(* CODESYS project OSCAT NETWORK.library
   Title: OSCAT NETWORK
   Author: Joel Zupancic
   Version: 1.30
   Description: see www.oscat.de for here home
      
      Made changes to use newer version 3 library SysSocket and SysFile.  All code was tested on CoDesys SoftPLC and Schneider Electric PLC with ehternet and file systems and using SoMachine software.
      
      
      IP_CONTROL
      1. Had to Set option for local address reuse in all network cases
        SysSockSetOption(socket, SOCKET_SOL, SOCKET_SO_REUSEADDR, ADR(dint_true), SIZEOF(dint_true));
      2. Had to change NETWORK_BUFFER_LONG_SIZE : UINT := 1999; //Changed from 3999 else socket would not work when reading 
      3. If PORT is zero use port specified by IP_C.C_PORT.
      4. CoDeSys has a bug that does not release the ports on a warm or cold reset.  What this means if you do a reset any function blocks that require binding to the socket to stay open will no longer work.  As of now the only way to clear the port is to recycle the power on the PLC.  
      
      
      TN_FRAMEWORK
      1.  Always Used Port 23. Changed to only use 23 if no port passed via IP_C.PORT
      
      STRING_TO_URL
      1.  Moved VAR_TEMP varible to VAR
      
      WORLD_WEATHER_ICON_OSCAT
      1.  Put [] around dat intial values
      
      YAHOO_WEATHER_ICON_OSCAT
      1.  Put [] around dat intial values
      
      MB_SERVER
      Need to reset the socket after the receive data timed out.  Since there is no code to detect that the Socket is still open you must force the socket closed and wait for the next connection.
      
      Case 10:
      IP_C.R_OBSERVE := TRUE; ( * keine Empfangsueberwachung * )
      
      and 
      
      IF ENABLE = FALSE OR t.Q THEN
          ip_state := BYTE#4; ( * Abmelden * )
         state := 00;
         IP_C.C_ENABLE := FALSE; 
      END_IF;
      
      
      /////////NEED TO FIX//////////////////
      FTP_CLIENT
      1.  Always Used Port 21. Changed to only use 21 if no port as specified in passed URL
   Company: OSCAT

Project tree, tasks and I/O mapping:
  libraries: SysTypes Interfaces, * (System); BASIC, 3.3.3.0 (OSCAT); Standard, * (System); SysSocket23, 3.5.8.0 (System); SysFile23, 3.5.8.0 (System)
  Data types/
    DATA_LOG/
      data type DLOG_CRON_DATA
      data type DLOG_CRON_ELEMENT
      data type DLOG_DATA
      data type DLOG_RETAIN
      data type LOG_CONTROL
      data type PRINTF_DATA
      data type UNI_CIRCULAR_BUFFER_DATA
      data type us_LOG_VIEWPORT
    DATABASE/
      data type MYSQL_COM
      data type MYSQL_INFO
    FILE_SERVER/
      data type FILE_PATH_DATA
      data type FILE_SERVER_DATA
    NET_VAR/
      data type NET_VAR_DATA
    NETWORK/
      data type IP2GEO_DATA
      data type IP_C
      data type IP_FIFO_DATA
      data type NETWORK_BUFFER
      data type NETWORK_BUFFER_SHORT
      data type NW_BUF_LONG
      data type NW_BUF_SHORT
      data type URL
      data type VMAP_DATA
      data type XML_CONTROL
    TELNET_VISION/
      data type us_TN_INPUT_CONTROL
      data type us_TN_INPUT_CONTROL_DATA
      data type us_TN_MENU
      data type us_TN_MENU_POPUP
      data type us_TN_SCREEN
    WEATHER/
      data type WORLD_WEATHER_CUR
      data type WORLD_WEATHER_DATA
      data type WORLD_WEATHER_DAY
      data type YAHOO_WEATHER_DATA
  Global Variables/
    global variables Constants
    global variables Globale_Variablen
  POUs/
    _HARDWARE/
      function block IP_CONTROL [ST]
      function block FILE_SERVER_OLD [ST]
      function block FILE_SERVER [ST]
      function block IP_CONTROL2 [ST]
    CONVERT/
      function block BASE64_DECODE_STR [ST]
      function block BASE64_DECODE_STREAM [ST]
      function block BASE64_ENCODE_STR [ST]
      function block BASE64_ENCODE_STREAM [ST]
      function HTML_DECODE [ST]
      function HTML_ENCODE [ST]
      function IP4_CHECK [ST]
      function IP4_DECODE [ST]
      function IP4_TO_STRING [ST]
      function IS_IP4 [ST]
      function IS_URLCHR [ST]
      function MD5_AUX [ST]
      function block MD5_CRAM_AUTH [ST]
      function block MD5_STR [ST]
      function block MD5_STREAM [ST]
      function MD5_TO_STRH [ST]
      function block RC4_CRYPT_STREAM [ST]
      function block SHA1_STR [ST]
      function block SHA1_STREAM [ST]
      function SHA1_TO_STRH [ST]
      function STRING_TO_URL [ST]
      function URL_DECODE [ST]
      function URL_ENCODE [ST]
      function URL_TO_STRING [ST]
    DATA_LOG/
      function block DLOG_BOOL [ST]
      function block DLOG_CRON_TAB [ST]
      function block DLOG_DINT [ST]
      function block DLOG_DT [ST]
      function block DLOG_FILE_TO_FTP [ST]
      function block DLOG_FILE_TO_SMTP [ST]
      function block DLOG_REAL [ST]
      function block DLOG_STORE_FILE_CSV [ST]
      function block DLOG_STORE_FILE_HTML [ST]
      function block DLOG_STORE_FILE_XML [ST]
      function block DLOG_STORE_MYSQL [ST]
      function block DLOG_STORE_RRD [ST]
      function block DLOG_STRING [ST]
      function block UNI_CIRCULAR_BUFFER [ST]
    DATABASE/
      function block MYSQL_AUTH [ST]
      function block MYSQL_CONTROL [ST]
    DRIVER/
      function block IRTRANS_DECODE [ST]
      function block IRTRANS_RCV_1 [ST]
      function block IRTRANS_RCV_4 [ST]
      function block IRTRANS_RCV_8 [ST]
      function block IRTRANS_SERVER [ST]
      function block IRTRANS_SND_1 [ST]
      function block IRTRANS_SND_4 [ST]
      function block IRTRANS_SND_8 [ST]
    FILE/
      function block CSV_PARSER_BUF [ST]
      function block CSV_PARSER_FILE [ST]
      function block FILE_BLOCK [ST]
      function FILE_PATH_SPLIT [ST]
      function block INI_PARSER_BUF [ST]
      function block INI_PARSER_FILE [ST]
    HARDWARE/
      function block FILE_SERVER_V2 [ST]
      function block IP_CONTROL_V2 [ST]
      function block IP_CONTROL2_V2 [ST]
    NET_VAR/
      function block NET_VAR_BOOL8 [ST]
      function block NET_VAR_BUFFER [ST]
      function block NET_VAR_CONTROL [ST]
      function block NET_VAR_DWORD8 [ST]
      function block NET_VAR_REAL8 [ST]
      function block NET_VAR_STRING [ST]
      function block NET_VAR_X8 [ST]
    NETWORK/
      function block DNS_CLIENT [ST]
      function block DNS_DYN [ST]
      function block DNS_REV_CLIENT [ST]
      function block FTP_CLIENT [ST]
      function block GET_WAN_IP [ST]
      function block HTTP_GET [ST]
      function block IP2GEO [ST]
      function block IP_FIFO [ST]
      function block LOG_MSG [ST]
      function block LOG_VIEWPORT [ST]
      function block MB_CLIENT [ST]
      function block MB_SERVER [ST]
      function block MB_SERVER_1 [ST]
      function block MB_VMAP [ST]
      function block PRINT_SF [ST]
      function block READ_HTTP [ST]
      function block SMTP_CLIENT [ST]
      function block SNTP_CLIENT [ST]
      function block SNTP_SERVER [ST]
      function block SPIDER_ACCESS [ST]
      function block SYS_LOG [ST]
      function block TELNET_LOG [ST]
      function block TELNET_PRINT [ST]
      function block XML_READER [ST]
    OTHER/
      function ELEMENT_COUNT [ST]
      function ELEMENT_GET [ST]
      function NETWORK_VERSION [ST]
    TELNET_VISION/
      function block TN_FRAMEWORK [ST]
      function block TN_INPUT_CONTROL [ST]
      function block TN_INPUT_EDIT_LINE [ST]
      function block TN_INPUT_MENU_BAR [ST]
      function block TN_INPUT_MENU_POPUP [ST]
      function block TN_INPUT_SELECT_POPUP [ST]
      function block TN_INPUT_SELECT_TEXT [ST]
      function block TN_RECEIVE [ST]
      function block TN_SC_ADD_SHADOW [ST]
      function block TN_SC_AREA_RESTORE [ST]
      function block TN_SC_AREA_SAVE [ST]
      function block TN_SC_BOX [ST]
      function block TN_SC_FILL [ST]
      function block TN_SC_LINE [ST]
      function block TN_SC_READ_ATTR [ST]
      function block TN_SC_READ_CHAR [ST]
      function TN_SC_SHADOW_ATTR [ST]
      function block TN_SC_VIEWPORT [ST]
      function block TN_SC_WRITE [ST]
      function block TN_SC_WRITE_ATTR [ST]
      function block TN_SC_WRITE_C [ST]
      function block TN_SC_WRITE_CHAR [ST]
      function block TN_SC_WRITE_EOS [ST]
      function TN_SC_XY2_ERROR [ST]
      function TN_SC_XY_ERROR [ST]
      function block TN_SEND_ROWS [ST]
    WEATHER/
      function block MOON_PHASE [ST]
      function block WORLD_WEATHER [ST]
      function block WORLD_WEATHER_DESC_GE [ST]
      function block WORLD_WEATHER_ICON_OSCAT [ST]
      function block YAHOO_WEATHER [ST]
      function block YAHOO_WEATHER_DESC_GE [ST]
      function block YAHOO_WEATHER_ICON_OSCAT [ST]
    DEMO/
      OLD/
        program INI_PARSER_FILE_DEMO_OLD [ST]
        program INI_PARSER_BUF_DEMO_OLD [ST]
      global variables GVL_DEMO
      Need Fixing/
        program IRTRANS_DEMO [CFC]
      WORKING/
        program INI_PARSER_BUF_DEMO [ST]
        program INI_PARSER_FILE_DEMO [ST]
        program _ECHO_TEST_DEMO [CFC]
        program CSV_PARSER_FILE_DEMO [ST]
        program TN_VISION_DEMO_1 [ST]
        program RC4_CRYPT_DEMO [CFC]
        program FILE_BLOCK_DEMO [CFC]
        program GET_WAN_IP_DEMO [CFC]
        program BASE64_DEMO [CFC]
        program DNS_SNTP_SYSLOG_DEMO [CFC]
        program DLOG_RRD_DEMO [CFC]
        program CSV_PARSER_BUF_DEMO [ST]
        program DNS_DYN_DEMO [CFC]
        program TN_VISION_DEMO_2 [ST]
        program YAHOO_WEATHER_DEMO [CFC]
        program MB_CLIENT_DEMO [CFC]
        program TELNET_LOG_DEMO [CFC]
        program SHA1_MD5_DEMO [CFC]
        program IP2GEO_DEMO [CFC]
        program FTP_CLIENT_DEMO [CFC]
        program MD5_CRAM_AUTH_DEMO [CFC]
        program DNS_CLEINT_DEMO [CFC]
        program TELNET_PRINT_DEMO [CFC]
        program HTTP_DEMO [CFC]
        program WORLD_WEATHER_DEMO [CFC]
        program MB_SERVER_DEMO [CFC]
        program SMTP_CLIENT_DEMO [CFC]
        program DNS_REV_DEMO [CFC]
      Need_Testing/
        program DLOG_FILE_CSV_FTP_DEMO [CFC]
        program DLOG_FILE_CSV_DEMO [CFC]
        program NET_VAR_SLAVE_DEMO [CFC]
        program DLOG_FILE_CSV_SMTP_DEMO [CFC]
        program SPIDER_DEMO [CFC]
        program DLOG_FILE_HTML_DEMO [CFC]
        program NET_VAR_MASTER_DEMO [CFC]
        program DLOG_MYSQL_DEMO [CFC]
        program DLOG_FILE_XML_DEMO [CFC]
  Visualizations/
*)

// Data types/DATA_LOG/DLOG_CRON_DATA
TYPE DLOG_CRON_DATA :
STRUCT
	CE : ARRAY [0..5] OF DLOG_CRON_ELEMENT;
END_STRUCT
END_TYPE

// Data types/DATA_LOG/DLOG_CRON_ELEMENT
TYPE DLOG_CRON_ELEMENT :
STRUCT
	ELEMENTS : ARRAY [0..59] OF BOOL;
	VALUE : INT;
	VALUE_MIN : INT;
	VALUE_MAX : INT;
	ALL_SELECTED : BOOL;
END_STRUCT
END_TYPE

// Data types/DATA_LOG/DLOG_DATA
TYPE DLOG_DATA :
STRUCT
	STORE_TYPE : BYTE;
	ADD_COM : INT;
	ADD_DATA_REQ : BOOL;
	CLOCK_TRIG : BOOL;
	ID_MAX : USINT;
	DTI : DT;
	UCB : UNI_CIRCULAR_BUFFER_DATA;
	LOAD_TIME_MAX : TIME;
	NEW_FILE : STRING;
	NEW_FILE_SIZE : UDINT;
	NEW_FILE_RTRIG : BOOL;
END_STRUCT
END_TYPE

(* revision history
ks	01. oct. 2010	rev 1.0
	original version

ks	13. may. 2011	rev 1.1
	neues Element: ADD_DATA_REQ

ks	26. jul. 2011	rev 1.2
	neues Element: STORE_TYPE

ks	16. apr. 2012	rev 1.3
	neues Elemente: NEW_FILE_SIZE, ADD_COM
*)

// Data types/DATA_LOG/DLOG_RETAIN
TYPE DLOG_RETAIN :
STRUCT
	FN_REM : STRING;
	COLOR : BOOL;
	HEAD: BOOL;
	TRIG_CNT : UDINT;
	TRIG_CNT_TOTAL : UDINT;
END_STRUCT
END_TYPE

(* revision history
ks	27. oct. 2012	rev 1.0
	original version

*)

// Data types/FILE_SERVER/FILE_PATH_DATA
TYPE FILE_PATH_DATA :
STRUCT
	DRIVE : STRING(3);
	DIRECTORY : STRING(OSCAT_BASIC.STRING_LENGTH);
	FILENAME : STRING;
END_STRUCT
END_TYPE

(* revision history
ks	01. oct. 2010	rev 1.0
	original version
*)

// Data types/FILE_SERVER/FILE_SERVER_DATA
TYPE FILE_SERVER_DATA :
STRUCT
	FILE_OPEN : BOOL;
	FILENAME : STRING;
	MODE : BYTE;
	OFFSET : UDINT;
	FILE_SIZE : UDINT;
	ERROR : BYTE;
END_STRUCT
END_TYPE

(* revision history
ks	05. mai. 2012	rev 1.1
	original version
*)

// Data types/NETWORK/IP2GEO_DATA
TYPE IP2GEO_DATA :
STRUCT
	STATE : BOOL;
	IP4 : DWORD;
	COUNTRY_CODE : STRING(2);
	COUNTRY_NAME : STRING(20);
	REGION_CODE : STRING(2);
	REGION_NAME : STRING(20);
	CITY : STRING(20);
	GEO_LATITUDE : REAL;
	GEO_LONGITUDE : REAL;
	TIME_ZONE_NAME : STRING(20);
	GMT_OFFSET : INT;
	IS_DST : BOOL;
END_STRUCT
END_TYPE

(* revision history
ks	14. aug. 2009	rev 1.0
	original version
*)

// Data types/NETWORK/IP_C
TYPE IP_C :
STRUCT
	C_MODE : BYTE;						(*W Mode: TCP/UCP AKTIV/PASSIV                               *)
	C_PORT : WORD;						(*W Portnummer                                               *)
	C_IP : DWORD;						(*W IP-Adresse gepackt wwxxyyzz = www.xxx.yyy.zzz            *)
	C_STATE : BYTE;						(*R Verbindungsstatus ON/OFF + Flanke ON/OFF                 *)
	C_ENABLE : BOOL;					(*W Freigabe für Connect                                     *)
	R_OBSERVE : BOOL;					(*W Empfang ueberwachen                                      *)
	TIME_RESET : BOOL;					(*W Alle Timer ruecksetzen                                   *)
	ERROR : DWORD;					(*R vvwwxxyy (vv = CON_ERROR, ww = SEN_ERROR, xx = REC_ERROR *)
	FIFO : IP_FIFO_DATA;					(*I IP FIFO Struktur                                         *)
	MAILBOX : ARRAY [1..16] OF BYTE;	(*I Mailbox: Datenbereich für Bausteindatenaustausch         *)
END_STRUCT
END_TYPE

(* revision history
ks	18. oct. 2008	rev 1.0
	original version
*)

// Data types/NETWORK/IP_FIFO_DATA
TYPE IP_FIFO_DATA :
STRUCT
	X : ARRAY [1..128] OF BYTE; 	(* IP_ID FIFO Speicher          *)
	Y : ARRAY [1..128] OF BYTE; 	(* IP_ID Zähler                 *)
	ID : BYTE;					(* höchste vergabene id         *)
	MAX_ID : BYTE;				(* maximal Anmeldungen pro ID   *)
	INIT : BOOL;					(* Initialisierung durchgeführt *)
	EMPTY : BOOL;				(* FIFO leer                    *)
	FULL : BOOL;					(* FIFO voll                    *)
	TOP : INT;					(* maximale anzahl in FIFO      *)
	NW : INT;					(* Schreibzeiger                *)
	NR : INT;						(* Lesezeiger                   *)
END_STRUCT
END_TYPE

(* revision history
ks	18. oct. 2008	rev 1.0
	original version
*)

// Data types/DATA_LOG/LOG_CONTROL
TYPE LOG_CONTROL :
STRUCT
	NEW_MSG : STRING(LOG_SIZE); (* neue Nachricht für den Datenbuffer *)
	NEW_MSG_OPTION : DWORD;
	LEVEL : BYTE;
	SIZE : INT := LOG_MAX; (* Anzahl der Strings im LOG_DATA *)
	RESET : BOOL; (* Nachrichtenbuffer löschen *)
	PRINTF : PRINTF_DATA; (* Array PRINTF Parameter *)
	MSG : ARRAY [0..LOG_MAX] OF STRING(LOG_SIZE); (* Array Message *)
	MSG_OPTION : ARRAY [0..LOG_MAX] OF DWORD; (* Array Options *)
	UPDATE_COUNT : UINT; (* Updatezähler *)
	IDX : INT; (* aktueller Nachrichten-Index *)
	RING_MODE : BOOL; (* Bufferüberlauf erkannt *)
END_STRUCT
END_TYPE

(* revision history
ks	18. oct. 2008	rev 1.0
	original version

ks	17..may. 2011	rev 1.1
	ENABLE entfernt

*)

// Data types/DATABASE/MYSQL_COM
TYPE MYSQL_COM :
STRUCT
	S_BUF : NETWORK_BUFFER;
	R_BUF : NETWORK_BUFFER;
	SQL_CON : BOOL;
	SQL_URL : STRING(OSCAT_BASIC.STRING_LENGTH);
	SQL_PACKET_NO : BYTE;
	TIMEOUT : TIME;
	DNS_IP4 : DWORD;
	SQL_RCV_STATE : BYTE;
	ERROR_C : DWORD;
	ERROR_T : BYTE;
END_STRUCT
END_TYPE

(* revision history
ks	27. oct. 2012	rev 1.0
	original version
*)

// Data types/DATABASE/MYSQL_INFO
TYPE MYSQL_INFO :
STRUCT
	SERVER_PROTOCOL_VERSION : BYTE;
	SERVER_CAPABILITIES : WORD;
	SERVER_STATUS : WORD;
	SERVER_LANGUAGE : BYTE;
	SQL_CONNECTED : BOOL;
	SQL_ERROR : STRING(OSCAT_BASIC.STRING_LENGTH);
END_STRUCT
END_TYPE

(* revision history
ks	27. oct. 2012	rev 1.0
	original version
*)

// Data types/NET_VAR/NET_VAR_DATA
TYPE NET_VAR_DATA :
STRUCT
	CYCLE : UDINT;
	STATE : BYTE;
	INDEX : INT;
	ID_MAX : USINT;
	ERROR_ID : BYTE;
	BUF_SIZE : UINT;
	S_BUF : NETWORK_BUFFER;
	R_BUF : NETWORK_BUFFER;
END_STRUCT
END_TYPE

(* revision history
ks	01. feb. 2011	rev 1.0
	original version
*)

// Data types/NETWORK/NETWORK_BUFFER
TYPE NETWORK_BUFFER :
STRUCT
	SIZE : UINT;
	BUFFER : NW_BUF_LONG;
END_STRUCT
END_TYPE

(* revision history
ks	01. 01. 2009	rev 1.0
	original version
*)

// Data types/NETWORK/NETWORK_BUFFER_SHORT
TYPE NETWORK_BUFFER_SHORT :
STRUCT
	SIZE : UINT;
	BUFFER : NW_BUF_SHORT;
END_STRUCT
END_TYPE

(* revision history
ks	01. 01. 2009	rev 1.0
	original version
*)

// Data types/NETWORK/NW_BUF_LONG
TYPE
	NW_BUF_LONG  : ARRAY[0..NETWORK_BUFFER_LONG_SIZE] OF BYTE;
END_TYPE

(* revision history
ks	01. 01. 2009	rev 1.0
	original version
*)

// Data types/NETWORK/NW_BUF_SHORT
TYPE
	NW_BUF_SHORT : ARRAY[0..NETWORK_BUFFER_SHORT_SIZE] OF BYTE;
END_TYPE

(* revision history
ks	01. 01. 2009	rev 1.0
	original version
*)

// Data types/DATA_LOG/PRINTF_DATA
TYPE PRINTF_DATA : ARRAY [1..11]  OF STRING(LOG_SIZE);
END_TYPE

(* revision history
ks	18. oct. 2008
	original version
*)

// Data types/DATA_LOG/UNI_CIRCULAR_BUFFER_DATA
TYPE UNI_CIRCULAR_BUFFER_DATA :
STRUCT
	D_MODE : INT;
	D_HEAD : WORD;
	D_STRING : STRING(OSCAT_BASIC.STRING_LENGTH);
	D_REAL : REAL;
	D_DWORD : DWORD;
	BUF_SIZE : UINT;
	BUF_COUNT : UINT;
	BUF_USED : USINT;
	BUF : NW_BUF_LONG;
	_GetStart : UINT;
	_GetEnd : UINT;
	_Last : UINT;
	_First : UINT;
END_STRUCT
END_TYPE

(* revision history
ks	01. oct. 2010	rev 1.0
	original version
*)

// Data types/NETWORK/URL
TYPE URL :
STRUCT
	PROTOCOL : STRING(10);
	USER : STRING(32);
	PASSWORD : STRING(32);
	DOMAIN : STRING(80);
	PORT : WORD;
	PATH : STRING(80);
	QUERY : STRING(OSCAT_BASIC.STRING_LENGTH);
	ANCHOR : STRING(40);
	HEADER : STRING(160);
END_STRUCT
END_TYPE

(* revision history
hm	18. oct. 2008 v1.0
	original version

ks	01.oct.2010 v1.1
	new header element and string size
*)

// Data types/DATA_LOG/us_LOG_VIEWPORT
TYPE us_LOG_VIEWPORT :
STRUCT
	LINE_ARRAY : ARRAY [1..40] OF INT;
	COUNT : INT; (* Anzahl der sichtbaren Nachtrichten *)
	UPDATE_COUNT : UINT; (* Updatezähler *)
	MOVE_TO_X : INT; (* Steuerung der Nachrichtenanzeige *)
	UPDATE : BOOL; (* Daten wurden geändert -> neuzeichnen *)
END_STRUCT
END_TYPE

(* revision history
ks	18. oct. 2008	rev 1.0
	original version
*)

// Data types/TELNET_VISION/us_TN_INPUT_CONTROL
TYPE us_TN_INPUT_CONTROL :
STRUCT
	bo_Enable: BOOL; (* Bearbeitung freigeben/sperren *)
	bo_Update_all: BOOL; (* All Elemente neu zeichnen *)
	bo_Reset_Fokus: BOOL; (* Fokus auf 1. Element setzen *)
	in_Focus_at: INT; (* Controlelement mit aktivem Fokus *)
	in_Count: INT; (* Anzahl der benutzen Control-Elemente *)
	in_ToolTip_X: INT; (* Tooltip Text X-Offset *)
	in_ToolTip_Y: INT; (* Tooltip Text Y-Offset *)
	by_ToolTip_Attr: BYTE; (* Tooltip Text Attribute *)
	in_ToolTip_Size: INT; (* Tooltip Text länge *)
	usa_TN_INPUT_CONTROL_DATA: ARRAY [1..20] OF us_TN_INPUT_CONTROL_DATA;
END_STRUCT
END_TYPE

(* revision history
ks	12. mai 2010	rev 1.0
	original version

*)

// Data types/TELNET_VISION/us_TN_INPUT_CONTROL_DATA
TYPE us_TN_INPUT_CONTROL_DATA :
STRUCT
 	by_Input_Exten_Code: BYTE;
	by_Input_ASCII_Code: BYTE;
	bo_Input_ASCII_IsNum: BOOL;
	in_Title_X_Offset: INT; (* Title Text X-Offset *)
	in_Title_Y_Offset: INT; (* Title Text Y-Offset *)
	by_Title_Attr: BYTE; (* Title Text Attribute *)
	st_Title_String: STRING; (* Title Text String *)
	in_Cursor_X: INT; (* aktuelle Cursor X-Position *)
	in_Cursor_Y: INT; (* aktuelle Cursor Y-Position *)
	in_Type: INT; (* Type des Elements *)
	in_X: INT; (* Element X-Position *)
	in_Y: INT; (* Element Y-Position *)
	in_Cursor_Pos: INT; (* aktuelle Cursorposition *)
	by_Attr_mF: BYTE; (* Text Attribute mit Fokus *)
	by_Attr_oF: BYTE; (* Text Attribute ohne Fokus *)
	in_selected: INT; (* Text Item wurde ausgewählt *)
	st_Input_Mask: STRING; (* Text Eingabemaske *)
	st_Input_Data: STRING(OSCAT_BASIC.STRING_LENGTH); (* Text aktuelle Eingabedaten *)
	st_Input_String: STRING; (* Text Kopie nach Return-Taste *)
	st_Input_ToolTip: STRING; (* Text ToolTip (Eingabeinformation) *)
	in_Input_Option: INT; (* Text Ausgabe-Optionen *)
	bo_Input_Entered: BOOL; (* RETURN-Taste wurde betätigt *)
	bo_Input_Hidden: BOOL; (* Text versteckete Eingabe mit '*' *)
	bo_Input_Only_Num: BOOL; (* Text nur Nummerneingabe zulassen *)
	bo_Focus: BOOL; (* Element besitzt den Fokus *)
	bo_Update_Input: BOOL; (* Element wegen Benutzereingabe neuzeichnen *)
	bo_Update_All: BOOL; (* Element komplett neuzeichnen *)

END_STRUCT
END_TYPE

(* revision history
ks	12. mai 2010	rev 1.0
	original version

*)

// Data types/TELNET_VISION/us_TN_MENU
TYPE us_TN_MENU :
STRUCT
	st_Menu_Text: STRING(OSCAT_BASIC.STRING_LENGTH); (* X Menue Texte *)
	in_Menu_E_Count: INT; (* Menue Elemente Anzahl *)
	in_Y: INT; (* Menue Zeilennummer  Y-Position *)
	in_X: INT; (* Menue Spaltennummer X-Position *)
	by_Attr_mF: BYTE; (* Text Attribute mit Fokus *)
	by_Attr_oF: BYTE; (* Text Attribute ohne Fokus *)
	in_X_SM_new: INT; (* neue Sub-Menu X-Position *)
	in_Y_SM_new: INT; (* neue Sub-Menu Y-Position *)
	in_X_SM_old: INT; (* alte Sub-Menu X-Position *)
	in_Y_SM_old: INT; (* alte Sub-Menu Y-Position *)
	in_Cur_Menu_Item: INT; (* aktuelles Haupt-Menue *)
	in_Cur_Sub_Item: INT; (* aktuelles Sub-Menue *)
	in_State: INT; (*   Menu status   *)
	in_Menu_Selected: INT; (* X Menu-Item mit Enter angewwählt *)
	bo_Create: BOOL; (* X Menu erzeugen *)
	bo_Destroy: BOOL; (* X Menu entfernen *)
	bo_Update: BOOL; (* X Menu updaten *)
END_STRUCT
END_TYPE

(* revision history
ks	12. mai 2010	rev 1.0
	original version

*)

// Data types/TELNET_VISION/us_TN_MENU_POPUP
TYPE us_TN_MENU_POPUP :
STRUCT
	st_Menu_Text: STRING(OSCAT_BASIC.STRING_LENGTH); (* X Menue Texte *)
	in_Menu_E_Count: INT; (* Menue Elemente Anzahl *)
	in_X: INT; (* X Menue X-Position *)
	in_Y: INT; (* X Menue Y-Position *)
	in_Cols: INT; (* Menue Spaltenanzahl *)
	in_Rows: INT; (* Menue Zeilenanzahl *)
	in_Cur_Item: INT; (* X aktuelles Sub-Menue *)
	by_Attr_mF: BYTE; (* X Text Attribute mit Fokus	*)
	by_Attr_oF: BYTE; (* X Text Attribute ohne Fokus *)
	by_Input_Exten_Code: BYTE; (* X Tastencode: Sondertasten *)
	bo_Create: BOOL; (* X Popup-Menu erzeugen *)
	bo_Destroy: BOOL; (* X Popup-Menu entfernen *)
	bo_Update: BOOL; (* X Popup-Menu updaten *)
	bo_Activ: BOOL; (*   Popup-Menu ist aktiv *)
END_STRUCT
END_TYPE

(* revision history
ks	12. mai 2010	rev 1.0
	original version

*)

// Data types/TELNET_VISION/us_TN_SCREEN
TYPE us_TN_SCREEN :
STRUCT
	bya_CHAR: ARRAY [0..1919] OF BYTE;
	bya_COLOR: ARRAY [0..1919] OF BYTE;
	bya_BACKUP: ARRAY [0..1919] OF BYTE;
	bya_Line_Update: ARRAY [0..23] OF BOOL;
	by_Input_Exten_Code: BYTE;
	by_Input_ASCII_Code: BYTE;
	bo_Input_ASCII_IsNum: BOOL;
	in_Page_Number: INT; (* aktive Seiten-Nr. *)
	in_Cursor_X: INT; (* Cursor X-Position *)
	in_Cursor_Y: INT; (* Cursor Y-Position *)
	in_EOS_Offset: INT; (* End of String Offset *)
	by_Clear_Screen_Attr: BYTE; (* Clear-Screen Attr *)
	bo_Clear_Screen: BOOL; (* Clear-Screen auslösen *)
	bo_Modal_Dialog: BOOL; (* Modaler Dialog ist aktiv *)
	bo_Menue_Bar_Dialog: BOOL; (* Menue Dialog ist aktiv *)
END_STRUCT
END_TYPE

(* revision history
ks	12. mai 2010	rev 1.0
	original version

*)

// Data types/NETWORK/VMAP_DATA
TYPE VMAP_DATA :
STRUCT
	FC : DWORD;
	V_ADR : INT;
	V_SIZE : INT;
	P_ADR : INT;
	TIME_OUT : TIME;
END_STRUCT
END_TYPE

(* revision history
ks	18. oct. 2008	rev 1.0
	original version
*)

// Data types/WEATHER/WORLD_WEATHER_CUR
TYPE WORLD_WEATHER_CUR :
STRUCT
	OBSERVATION_TIME : STRING(8);
	TEMP_C : INT;
	WEATHER_CODE : INT;
	WEATHER_DESC : STRING(60);
	WEATHER_ICON : INT;
	WIND_SPEED_MILES : INT;
	WIND_SPEED_KMPH : INT;
	WIND_DIR_DEGREE : INT;
	WIND_DIR16POINT : STRING(3);
	PRECIPMM : REAL;
	HUMIDITY : INT;
	VISIBILITY : INT;
	PRESSURE : INT;
	CLOUDOVER : INT;
END_STRUCT
END_TYPE

(* revision history
ks	01. oct. 2010	rev 1.0
	original version

ks	04. may. 2011	rev 1.1
	neues element:  WEATHER_ICON


*)

// Data types/WEATHER/WORLD_WEATHER_DATA
TYPE WORLD_WEATHER_DATA :
STRUCT
	CUR : WORLD_WEATHER_CUR;
	DAY : ARRAY [0..4] OF WORLD_WEATHER_DAY;
END_STRUCT
END_TYPE

(* revision history
ks	01. oct. 2010	rev 1.0
	original version

*)

// Data types/WEATHER/WORLD_WEATHER_DAY
TYPE WORLD_WEATHER_DAY :
STRUCT
	DATE_OF_DAY : STRING(10);
	TEMP_MAX_C : INT;
	TEMP_MAX_F : INT;
	TEMP_MIN_C : INT;
	TEMP_MIN_F : INT;
	WIND_SPEED_MILES : INT;
	WIND_SPEED_KMPH : INT;
	WIND_DIR_DEGREE : INT;
	WIND_DIR16POINT : STRING(3);
	WEATHER_CODE : INT;
	WEATHER_DESC : STRING(60);
	WEATHER_ICON : INT;
	PRECIPMM : REAL;
END_STRUCT
END_TYPE

(* revision history
ks	01. oct. 2010	rev 1.0
	original version

ks	04. may. 2011	rev 1.1
	neues element:  WEATHER_ICON


*)

// Data types/NETWORK/XML_CONTROL
TYPE XML_CONTROL :
STRUCT
	COMMAND : WORD;
	WATCHDOG : TIME;
	START_POS : UINT;
	STOP_POS : UINT;
	COUNT : UINT;
	TYP : INT;
	LEVEL : UINT;
	PATH : STRING(OSCAT_BASIC.STRING_LENGTH);
	ELEMENT : STRING(OSCAT_BASIC.STRING_LENGTH);
	ATTRIBUTE : STRING(OSCAT_BASIC.STRING_LENGTH);
	VALUE : STRING(OSCAT_BASIC.STRING_LENGTH);
	BLOCK1_START : UINT;
	BLOCK1_STOP : UINT;
	BLOCK2_START : UINT;
	BLOCK2_STOP : UINT;
END_STRUCT
END_TYPE

(* revision history
ks	18. oct. 2008	rev 1.0
	original version

ks	24. sep. 2010	rev 1.1
	STRING(STRING_LENGTH)
*)

// Data types/WEATHER/YAHOO_WEATHER_DATA
TYPE YAHOO_WEATHER_DATA :
STRUCT
	TIMETOLIVE : INT;							(* TIME TO LIVE: HOW LONG IN MINUTES THIS FEED SHOULD BE CACHED         *)
	LOCATION_CITY : STRING(40);   				(* THE LOCATION OF THIS FORECAST: CITY: CITY NAME  *)
	LOCATION_REGION : STRING(20);  				(* THE LOCATION OF THIS FORECAST: REGION: STATE, TERRITORY, OR REGION, IF GIVEN *)
	LOCATION_COUNTRY : STRING(20);			(* THE LOCATION OF THIS FORECAST: COUNTRY: TWO-CHARACTER COUNTRY CODE *)
	UNIT_TEMPERATURE : STRING(1);				(* TEMPERATURE: DEGREE UNITS, F FOR FAHRENHEIT OR C FOR CELSIUS *)
	UNIT_DISTANCE : STRING(2);					(* DISTANCE: UNITS FOR DISTANCE, MI FOR MILES OR KM FOR KILOMETERS *)
	UNIT_PRESSURE : STRING(2);					(* PRESSURE: UNITS OF BAROMETRIC PRESSURE, IN FOR POUNDS PER SQUARE INCH OR MB FOR MILLIBARS *)
	UNIT_SPEED : STRING(4);						(* SPEED: UNITS OF SPEED, MPH FOR MILES PER HOUR OR KPH FOR KILOMETERS PER HOUR *)
	WIND_CHILL : INT;							(* FORECAST INFORMATION ABOUT WIND CHILL IN DEGREES *)
	WIND_DIRECTION : INT;						(* FORECAST INFORMATION ABOUT WIND DIRECTION, IN DEGREES *)
	WIND_SPEED : REAL;							(* FORECAST INFORMATION ABOUT WIND SPEED, IN THE UNITS (MPH OR KPH)*)
	ATMOSPHERE_HUMIDITY : INT;				(* FORECAST INFORMATION ABOUT CURRENT ATMOSPHERIC HUMIDITY: HUMIDITY, IN PERCENT  *)
	ATMOSPHERE_PRESSURE : INT;				(* FORECAST INFORMATION ABOUT CURRENT ATMOSPHERIC PRESSURE: BAROMETRIC PRESSURE, IN THE UNITS (IN OR MB) *)
	ATMOSPHERE_VISIBILITY : REAL;				(* FORECAST INFORMATION ABOUT CURRENT ATMOSPHERIC VISIBILITY, IN THE UNITS (MI OR KM) *)
	ATMOSPHERE_RISING : INT;					(* FORECAST INFORMATION ABOUT RISING: STATE OF THE BAROMETRIC PRESSURE: STEADY (0), RISING (1), OR FALLING (2). (INTEGER: 0, 1, 2) *)
	ASTRONOMY_SUNRISE : STRING(10);			(* SUNRISE: TODAY'S SUNRISE TIME. THE TIME IS A STRING IN A LOCAL TIME FORMAT OF "H:MM AM/PM" *)
	ASTRONOMY_SUNSET : STRING(10);			(* SUNSET: TODAY'S SUNSET TIME. THE TIME IS A STRING IN A LOCAL TIME FORMAT OF "H:MM AM/PM", *)
	GEO_LATITUDE : REAL;						(* THE LATITUDE OF THE LOCATION *)
	GEO_LONGITUDE : REAL;						(* THE LONGITUDE OF THE LOCATION *)
	CUR_CONDITIONS_TEMP : INT;				(* THE CURRENT WEATHER CONDITIONS: TEMP: THE CURRENT TEMPERATURE, IN THE UNITS (F OR C) *)
	CUR_CONDITIONS_TEXT : STRING(40);			(* THE CURRENT WEATHER CONDITIONS: TEXT: A TEXTUAL DESCRIPTION OF CONDITIONS *)
	CUR_CONDITIONS_CODE : INT;				(* THE CURRENT WEATHER CONDITIONS: CODE: THE CONDITION CODE FOR THIS FORECAST *)
	CUR_CONDITIONS_ICON : INT;					(* THE CURRENT WEATHER CONDITIONS: ICON: THE CONDITION ICON FOR THIS FORECAST *)
	FORCAST_TODAY_LOW_TEMP : INT;			(* THE FORCAST TODAY WEATHER CONDITIONS: THE FORECASTED LOW TEMPERATURE FOR THIS DAY IN THE UNITS (F OR C) *)
	FORCAST_TODAY_HIGH_TEMP : INT;			(* THE FORCAST TODAY WEATHER CONDITIONS: THE FORECASTED HIGH TEMPERATURE FOR THIS DAY IN THE UNITS (F OR C) *)
	FORCAST_TODAY_TEXT : STRING(40);			(* THE FORCAST TODAY WEATHER CONDITIONS: TEXT: A TEXTUAL DESCRIPTION OF CONDITIONS *)
	FORCAST_TODAY_CODE : INT;				(* THE CURRENT WEATHER CONDITIONS: CODE: THE CONDITION CODE FOR THIS FORECAST *)
	FORCAST_TODAY_ICON : INT;					(* THE CURRENT WEATHER CONDITIONS: ICON: THE CONDITION ICON FOR THIS FORECAST *)
	FORCAST_TOMORROW_LOW_TEMP : INT; 		(* THE FORCAST TOMORROW WEATHER CONDITIONS: THE FORECASTED LOW TEMPERATURE FOR THIS DAY IN THE UNITS (F OR C) *)
	FORCAST_TOMORROW_HIGH_TEMP : INT;		(* THE FORCAST TOMORROW WEATHER CONDITIONS: THE FORECASTED HIGH TEMPERATURE FOR THIS DAY IN THE UNITS (F OR C) *)
	FORCAST_TOMORROW_TEXT : STRING(40);	(* THE FORCAST TOMORROW WEATHER CONDITIONS: TEXT: A TEXTUAL DESCRIPTION OF CONDITIONS *)
	FORCAST_TOMORROW_CODE : INT;			(* THE CURRENT WEATHER CONDITIONS: CODE: THE CONDITION CODE FOR THIS FORECAST *)
	FORCAST_TOMORROW_ICON : INT;			(* THE CURRENT WEATHER CONDITIONS: ICON: THE CONDITION ICON FOR THIS FORECAST *)

END_STRUCT
END_TYPE

(* revision history
ks	18. oct. 2008	rev 1.0
	original version

ks	24. sep. 2010	rev 1.1
	LOCATION_COUNTRY STRING(20)

ks	04. may. 2011	rev 1.2
	neue elemente:  CUR_CONDITIONS_ICON, FORCAST_TODAY_ICON, FORCAST_TOMORROW_ICON
*)

// Global Variables/Constants
VAR_GLOBAL CONSTANT
	//NETWORK_BUFFER_LONG_SIZE : UINT := 4095;
	NETWORK_BUFFER_LONG_SIZE : UINT := 1999;
	NETWORK_BUFFER_SHORT_SIZE : UINT := 1407;
	LOG_MAX : INT := 40;
	LOG_SIZE : INT := 80;
	ELEMENT_LENGTH : INT := 250;
END_VAR

// Global Variables/Globale_Variablen
VAR_GLOBAL
	(* ------- only for Beckhoff - TwinCat  --------- *)
	TCP_SERVER_RESET : BYTE; (* only for internaly use - do't modify *)
	sSrvNetId : STRING(23) := ''; (* String containing the network address of the TwinCAT TCP/IP Connection Server (e.g. '1.1.1.2.7.1'). For the local computer (default) an empty string may be specified *)
	sLocalHost : STRING(15) := ''; (* The local IP address (Ipv4) of the UDP client/server socket as a string (e.g. '172.33.5.1'). An empty string may be specified for the default network adapter *)
	(* --------------------------------------------- *)

	(* ------- only for CoDeSys -------------------- *)
	SYSLIBSOCKETS_OPTION : BYTE := BYTE#2#0000_0000;	(* Configuration option for SysLibSocket.lib / Bit 0 = 1 -> TCP-Client - SysSockselect for PLCWinNT *)
	(* --------------------------------------------- *)

	LOG_CL : LOG_CONTROL;
END_VAR

// POUs/DEMO/GVL_DEMO
VAR_GLOBAL
	smtp_server: STRING;
	smtp_mailfrom: STRING ;
	smtp_mailto: STRING;
		
    //Default Google Public DNS
	DNS_IP_OCTET_3: BYTE := 8;
	DNS_IP_OCTET_2: BYTE := 8;
	DNS_IP_OCTET_1: BYTE := 8;
	DNS_IP_OCTET_0: BYTE := 8;
	
	ftp_url: STRING;
END_VAR

// POUs/_HARDWARE/IP_CONTROL
FUNCTION_BLOCK IP_CONTROL
VAR_IN_OUT
	IP_C : IP_C; (* IP_Control Verwaltungsstruktur *)
	S_BUF : NETWORK_BUFFER; (* Externer Sendbuffer *)
	R_BUF : NETWORK_BUFFER; (* Externer Receivebuffer *)
END_VAR
VAR_INPUT
	IP : DWORD; (* IP Adresse *)
	PORT : WORD; (* Port Nummer *)
	TIME_OUT : TIME; (* Ueberwachungszeit Connect / Send / Receive *)
END_VAR
VAR
	c_time : UDINT; (* CONNECT-Time (Zeit bei nicht vorhandener Verbindung) *)
	s_time : UDINT; (* SEND-Time    (Zeit seit letzten Datensenden) *)
	r_time : UDINT; (* RECEIVE-Time (Zeit seit letztem Datenempfang) *)

	c_enable : BOOL; (* Connect: freigabe *)
	c_ip : DWORD; (* Connect: aktuelle IP-Adresse *)
	c_port : WORD; (* Connect: aktuelle Port-Nummer *)
	c_mode : BYTE; (* Connect: aktueller Mode UDP/TCP...... *)
	c_status : BYTE; (* Connect: Status (Errorcode) *)
	c_ready : BOOL; (* Connect: Verbindung aufgebaut *)
	c_ready_old : BOOL; (* Connect: letzter Zustand von c_ready für Flankenauswertung *)
	c_select : BOOL; (* non blocking mode - abfrage über select durchführen *)
	c_fdWrite : SOCKET_FD_SET;
	c_Timeout : SOCKET_TIMEVAL;

	s_total : INT; (* Send: Gesamtanzahl Bytes zum senden *)
	s_cur_pos : INT; (* Send: aktuelle Sendeposition *)
	s_cur_size : INT; (* Send: aktuelle Sendegroesse *)
	s_max_size : INT; (* Send: maximale Telegrammlänge fuer Senden *)
	s_start : BOOL; (* Send: Sende modus aktivieren *)
	s_active : BOOL; (* Send: Daten senden ist aktiv *)
	s_req : BOOL; (* Send: Start Daten senden *)
	s_done : BOOL; (* Send: ohne Fehler beendet *)
	s_status : BYTE; (* Send: Status (Errorcodes) *)

	r_status : BYTE; (* Receive: Status (Errorcodes) *)
	r_count : INT; (* Receive: Anzahl empfangener Bytes *)
	r_offset : INT; (* Receive: aktuelle Position in externen Receivebuffer *)
	r_max_size : INT; (* Receive: groesse des externen Empfangbuffers*)

	new_connection : BOOL; (* Neue Verbindungsparameter vorhanden *)
	tx : DWORD; (* letzter zeitwert *)
	error_time : DWORD; (* aktueller Timeout-Wert *)

	state: BYTE; (* schrittmerker für connect *)
	server_socket : RTS_IEC_HANDLE:= RTS_INVALID_HANDLE;                // Handle Pointing to our Socket
	socket : RTS_IEC_HANDLE:= RTS_INVALID_HANDLE;
	//server_socket : DINT:= RTS_INVALID_HANDLE;
	//socket : DINT:= RTS_INVALID_HANDLE;
	sockaddr : SOCKADDRESS;
	sockaddr_size : DWORD;
	plc_841 : BOOL;
	plc_881 : BOOL;
	dint_true : DINT := 1;
	bytes_received : DINT;
	bytes_sent : DINT;
	udp_mode : BOOL;

	pResult : UDINT; //Needed for V3 Lib
	FunctionResult 	: UDINT ;   
  	tAddress                	: INADDR;                           // Strucutre to define our internet address
	TESTtAddress               	: INADDR;   
	(*LOG_MSG : LOG_MSG;
	_debug_enable : BOOL := TRUE;
	debug_index : INT;
	debug_ID : INT;
	debug_lasterror : DWORD;
	debug_last_id : INT := 255;
	state_last: BYTE;*)

END_VAR

VAR CONSTANT
	STOP : BYTE := 0;
	TS_INIT: BYTE := 1;
	TS_OPEN : BYTE:= 2;

	UDP_INIT : BYTE:= 31;

	TC_INIT : BYTE:= 51;
	TC_CONNECT : BYTE:= 52;

	C_WAIT : BYTE:= 250;
	C_CLOSE : BYTE:= 251;

END_VAR

(*

version 1.9		26. Feb. 2012
programmer 		ks
tested by			ks

IP_CONTROL ist ein Wrapper-Baustein um eine Hersteller neutrale Schnittstelle zum Ethernet zu schaffen
*)

(* ---------------------- Debug-Message ----------------------------*)
(*IF _debug_enable THEN
	IF IP_C.FIFO.ID > BYTE#0 THEN (* nur wenn Teilnehmer ID's vorhanden sind *)
		debug_index := IP_C.FIFO.NR;
		debug_ID := BYTE_TO_INT(IP_C.FIFO.X[debug_index]);
	END_IF;
END_IF;*)
(* -----------------------------------------------------------------------------*)

(* read system time *)
tx := T_PLC_MS();

IF IP_C.C_PORT = 0 THEN
	IP_C.C_PORT := PORT; (* uebergebenen PORT durch parametrierten PORT ersetzen *)
END_IF;
IF IP_C.C_IP = 0 AND IP_C.C_MODE < 4 THEN
	IP_C.C_IP := IP; (* uebergebene IP durch paramtrierte IP ersetzen *)
END_IF;

new_connection := c_ip <> IP_C.C_IP OR c_mode <> IP_C.C_MODE OR c_port <> IP_C.C_PORT; (* neue Verbindungs erwünscht ? *)
c_enable := IP_C.C_ENABLE AND NOT new_connection;

IF IP_C.C_ENABLE AND IP_C.ERROR = 0 AND state = STOP THEN (* Freigabe,kein Fehler,kein Socket offen *)
	c_ip   := IP_C.C_IP;
	c_mode := IP_C.C_MODE;
	c_port := IP_C.C_PORT;
	plc_841 := ADR(%MW0)=16#30000000; (*750-841*)
	plc_881 := ADR(%MW0)=16#20000000; (*750-881*)
	udp_mode := C_MODE.0; (* Mode 1,3,5 = udp *)

	error_time := TIME_TO_DWORD(MAX(T#200ms,TIME_OUT));
	IP_C.TIME_RESET := TRUE; (* Alle Timer ruecksetzen *)

	r_max_size := UINT_TO_INT(SIZEOF(R_BUF.BUFFER));
	s_max_size := UINT_TO_INT(SIZEOF(S_BUF.BUFFER));

	IF C_MODE.0 THEN (* Mode: 1,3,5 = UDP CLIENT/SERVER *)
		state := UDP_INIT;
	ELSIF C_MODE = 0 THEN (* Mode: 0 = TCP CLIENT *)
		state := TC_INIT;
	ELSE
		state := TS_INIT; (* Mode: 2,4 = TCP SERVER *)
	END_IF;

	(* ---------------------- Debug-Message ----------------------------*)
	(*IF _debug_enable THEN
		LOG_CL.NEW_MSG := 'IP_CON: MODE ~1 / IP ~2 / PORT ~3 /ID ~6';
		LOG_CL.PRINTF[1] := BYTE_TO_STRING(C_MODE);
		LOG_CL.PRINTF[2] := IP4_TO_STRING(c_ip);
		LOG_CL.PRINTF[3] := WORD_TO_STRING(c_port);
		LOG_CL.PRINTF[6] := INT_TO_STRING(debug_ID);
		LOG_MSG();
	END_IF;*)
	(* -----------------------------------------------------------------------------*)

END_IF;

(* ---------------------- Debug-Message ----------------------------*)
(*IF  _debug_enable THEN
	IF state <> state_last THEN
		LOG_CL.NEW_MSG := 'IP_STEP ~1 -IP_ID ~6';
		LOG_CL.PRINTF[1] := BYTE_TO_STRING(state);
		LOG_CL.PRINTF[6] := INT_TO_STRING(debug_ID);
		LOG_MSG();
		state_last := state;
	END_IF;
END_IF;*)
(* -----------------------------------------------------------------------------*)

IF IP_C.TIME_RESET THEN (* Alle Timer ruecksetzen *)
	IP_C.TIME_RESET := FALSE; (* Reset rücksetzen *)
	c_time := tx; (* Connect Timer ruecksetzen *)
	s_time := tx; (* Send Timer ruecksetzen *)
	r_time := tx; (* Receive Timer ruecksetzen *)

	c_status := BYTE#0; (* letzten Connect Fehler rücksetzen *)
	s_status := BYTE#0; (* letzten Send Fehler rücksetzen *)
	r_status := BYTE#0; (* letzten Receive Fehler rücksetzen *)
END_IF;

(* ---------------------------------------------- *)

CASE state OF

UDP_INIT: (* UDP_CLIENT + SERVER *)
	socket := SysSockCreate(SOCKET_AF_INET, SOCKET_DGRAM, SOCKET_IPPROTO_IP, ADR(pResult));
	IF socket < 0 THEN
		c_status := 1; (* SysSockCreate failed *)
		state := C_CLOSE;
	ELSE
		FunctionResult :=SysSockSetOption(socket, SOCKET_SOL, SOCKET_SO_BROADCAST, ADR(dint_true), SIZEOF(dint_true)); (* allow broadcast *)
		FunctionResult :=SysSockIoctl(socket, SOCKET_FIONBIO, ADR(dint_true)); (* put socket in non-blocking mode *)
		sockaddr.sin_family := SOCKET_AF_INET;
		sockaddr.sin_port := SysSockHtons(c_port);
		sockaddr.sin_addr.ulAddr := SEL(c_mode = 1, SOCKET_INADDR_ANY, SysSockNtohl(c_ip));

		IF c_mode >= 2 THEN (* SERVER Mode *)
			FunctionResult := SysSockBind(socket, ADR(sockaddr), SIZEOF(sockaddr));
			IF FunctionResult=0 THEN
				c_ready := TRUE; (* Connected *)
				state:= C_WAIT;
			ELSE
				c_status := 2; (* SysSockBind failed *)
				state := C_CLOSE;
			END_IF;
		ELSE
			c_ready := TRUE; (* Connected *)
			state:= C_WAIT;
		END_IF;
	END_IF;

(* ---------------------------------------------- *)

TC_INIT: (* TCP-CLIENT (AKTIV) *)
	// Create handle to ethernet socket to send messages
	socket        := SysSockCreate(SOCKET_AF_INET, SOCKET_STREAM, SOCKET_IPPROTO_TCP, ADR(pResult)); 	
	IF socket < 0 THEN
		c_status := 1;  (* SysSockCreate failed *)
		state := C_CLOSE;
	ELSE
		IF plc_841 OR plc_881 THEN
			FunctionResult :=SysSockSetOption(socket,6,SOCKET_TCP_NODELAY, ADR(dint_true), SIZEOF(dint_true)); (* Set Push-Bit *)
		END_IF;
		// Set option for local address reuse
		FunctionResult :=SysSockSetOption(socket, SOCKET_SOL, SOCKET_SO_REUSEADDR, ADR(dint_true), SIZEOF(dint_true));
		// Set option for keepalive
		//FunctionResult := SysSockSetOption(socket, SOCKET_SOL, SOCKET_SO_KEEPALIVE, ADR(dint_true), SIZEOF(dint_true));
		
        //Moved to After Connect 
		//FunctionResult :=SysSockIoctl(socket, SOCKET_FIONBIO, ADR(dint_true)); (* NonBlocking mode *)
		
		sockaddr.sin_family := SOCKET_AF_INET;
		sockaddr.sin_port := SysSockNtohs(c_port);
		sockaddr.sin_addr.ulAddr  := SysSockNtohl(c_ip);
		c_select := FALSE;
		state := TC_CONNECT;
	END_IF;

(* ---------------------------------------------- *)

TC_CONNECT:
	IF NOT c_enable OR c_status = 255 THEN (* keine freigabe oder connect timeout *)
			state:= C_CLOSE;
	ELSE
		IF c_select = FALSE THEN
			FunctionResult:=SysSockConnect(socket,ADR(sockaddr),SIZEOF(sockaddr));
			IF FunctionResult=0 THEN
				FunctionResult :=SysSockIoctl(socket, SOCKET_FIONBIO, ADR(dint_true)); (* NonBlocking mode *)
				c_ready := TRUE; (* Connected *)
				state:= C_WAIT;
			ELSE
				(* Connect durchgeführt, aber noch nicht verbunden, dann optional mit select-abfrage weitermachen *)
				c_select := SYSLIBSOCKETS_OPTION.0; (* Bit 0 = TCP-Client - use SysSockselect *)
			END_IF;
		ELSE
			c_Timeout.tv_sec := 0;
			c_Timeout.tv_usec := 0;
			c_fdWrite.fd_count := 1;
			c_fdWrite.fd_array[0] := socket;
			IF SysSockSelect(SOCKET_FD_SETSIZE,0,ADR(c_fdWrite),0, ADR(c_Timeout), ADR(pResult)) > 0 THEN
				c_ready := TRUE; (* Connected *)
				state:= C_WAIT;
			END_IF;
		END_IF;
	END_IF;

(* ---------------------------------------------- *)

TS_INIT: (* TCP-SERVER (PASSIV) *)
	server_socket := SysSockCreate(SOCKET_AF_INET, SOCKET_STREAM, SOCKET_IPPROTO_IP, ADR(pResult)); (* Create Socket *)
	IF server_socket = RTS_INVALID_HANDLE THEN
		c_status := 1; (* SysSockCreate failed *)
		state:= C_CLOSE;
	ELSE (* Address bindings *)
		SysSockSetOption( server_socket, SOCKET_SOL, SOCKET_SO_REUSEADDR, ADR(dint_true), SIZEOF(dint_true) );
		sockaddr.sin_family:= SOCKET_AF_INET;
		sockaddr.sin_port := SysSockHtons(c_port);
		sockaddr.sin_addr.ulAddr  := SOCKET_INADDR_ANY;
		IF NOT SysSockBind(server_socket, ADR(sockaddr), SIZEOF(sockaddr)) = 0 THEN
			c_status := 2; (* SysSockBind failed *)
			state := C_CLOSE;
		ELSIF NOT SysSockListen(server_socket, 1) = 0 THEN (* erzeugt Warteschlange für eine Verbindung *)
			c_status := 3; (* SysSockListen failed *)
			state:= C_CLOSE;
		ELSE
			SysSockIoctl(server_socket, SOCKET_FIONBIO, ADR(dint_true)); (* NonBlocking mode *)
			state:= TS_OPEN;
		END_IF;
	END_IF;

(* ---------------------------------------------- *)

TS_OPEN: (* Waiting for incomming connection *)
	sockaddr_size := SIZEOF(sockaddr);
	socket := SysSockAccept(server_socket, ADR(sockaddr), ADR(sockaddr_size), ADR(pResult));

	IF socket <> RTS_INVALID_HANDLE THEN (* neuer Verbindungswunsch vorhanden *)
		IF c_mode = BYTE#2 AND sockaddr.sin_addr.ulAddr <> SysSockNtohl(c_ip) THEN (* Mode 2 = TCP + PASSIVE + PORT + IP  auf richtige Partner-IP prüfen *)
			state:= C_CLOSE;
		ELSE
			IF plc_841 OR plc_881 THEN
				SysSockSetOption(socket, 6, SOCKET_TCP_NODELAY, ADR(dint_true), SIZEOF(dint_true)); (* Set Push-Bit *)
			END_IF;
			SysSockIoctl(socket, SOCKET_FIONBIO, ADR(dint_true)); (* NonBlocking mode *)
			c_ready := TRUE; (* Connected *)
			state := C_WAIT;
		END_IF;
	ELSIF NOT c_enable THEN (* keine freigabe mehr ? *)
			state:= C_CLOSE;
	END_IF;

(* ---------------------------------------------- *)

C_WAIT: (* Warten auf Anforderung für Beenden *)
	IF NOT c_enable OR NOT c_ready THEN
		state:= C_CLOSE;
	END_IF

(* ---------------------------------------------- *)

C_CLOSE: (* Close the Sockets *)
	c_ready := FALSE;
	IF socket >= 0 THEN
		IF (NOT plc_841) AND (NOT plc_881) THEN
			SysSockShutdown(socket, 0); (* 870 *)
		END_IF;
		SysSockClose(socket);
		socket := RTS_INVALID_HANDLE;
	END_IF
	IF server_socket >= 0 THEN
		IF (NOT plc_841) AND (NOT plc_881) THEN
			SysSockShutdown(server_socket, 0); (* 870 *)
		END_IF;
		SysSockClose(server_socket);
		server_socket := RTS_INVALID_HANDLE;
	END_IF
	state:= STOP;
END_CASE;

(* ---------------------------------------------- *)

IF c_ready THEN
	IF NOT c_ready_old THEN (* Verbindung aufgebaut - positive Flanke erkannt *)
		IP_C.C_STATE := 254;
		IP_C.TIME_RESET := TRUE; (* Alle Timer ruecksetzen *)
		(* ---------------------- Debug-Message ----------------------------*)
		(*IF _debug_enable THEN
			LOG_CL.NEW_MSG := 'IP_CON: CONNECTED -IP_ID ~6';
			LOG_CL.PRINTF[6] := INT_TO_STRING(debug_ID);
			LOG_MSG();
		END_IF;*)
		(* -----------------------------------------------------------------------------*)
	ELSE
		IP_C.C_STATE := 255; (* Verbindung ist aufgebaut *)
	END_IF;
ELSE
	IF c_ready_old THEN (* Verbindung abgebaut - negative Flanke erkannt *)
		IP_C.C_STATE := 1;
		IP_C.MAILBOX[1] := 0; (* Receive Info rücksetzen *)
		IP_C.MAILBOX[2] := 0; (* Send-Pause rücksetzen *)
		IP_C.MAILBOX[3] := 0; (* Receive-Pause rücksetzen *)
		IF NOT new_connection THEN
			s_active := FALSE; (* Sendeaktivitäten stoppen *)
			s_req := FALSE; (* Sendefreigabe rücksetzen *)
			S_BUF.SIZE := 0; (* Sendelänge löschen *)
			(*IP_C.TIME_RESET := TRUE;*) (* Alle Timer ruecksetzen *)
		END_IF;
		(* ---------------------- Debug-Message ----------------------------*)
		(*IF _debug_enable THEN
			LOG_CL.NEW_MSG := 'IP_CON: DISCONNECTED';
			LOG_MSG();
		END_IF;*)
		(* -----------------------------------------------------------------------------*)
	ELSE
		IP_C.C_STATE := 0; (* Verbindung ist abgebaut *)
	END_IF;
END_IF;

c_ready_old := c_ready;

(* Der Datenempfang wird angehalten solange ein Sendevorgang läuft *)
(* sonst kann es vorkommen das die Antwort-daten schon empfangen werden, *)
(* bevor der Sendevorgang vom programm abgeschlossen wurde *)

IF c_ready AND NOT s_active AND IP_C.MAILBOX[3] = 0 THEN
	IF R_BUF.SIZE >= INT_TO_UINT(r_max_size) THEN
		R_BUF.SIZE := UINT#0;
		r_status := 254; (* Empfangsbuffer wegen Überlauf rückgesetzt *)
	END_IF;

	r_offset := SEL(udp_mode,UINT_TO_INT(R_BUF.SIZE),0);
	r_count := r_max_size - r_offset;

	IF udp_mode THEN
		bytes_received := SysSockRecvFrom(socket, ADR(R_BUF.BUFFER), r_count, 0, ADR(sockaddr), SIZEOF(sockaddr), ADR(pResult));

		IF c_mode = BYTE#3 AND sockaddr.sin_addr.ulAddr <> SysSockNtohl(c_ip) THEN (* Mode 3 = UDP + PASSIVE + PORT + IP  auf richtige Partner-IP prüfen *)
			bytes_received := 0;
			R_BUF.SIZE := UINT#0;
			sockaddr.sin_port := SysSockNtohs(c_port);
			sockaddr.sin_addr.ulAddr  := SysSockNtohl(c_ip);
		END_IF;

	ELSE
		bytes_received := SysSockRecv(socket, ADR(R_BUF.BUFFER[r_offset]), r_count, 0, ADR(pResult));
	END_IF;

	CASE pResult OF
		518:  bytes_received:=-1; //Connection OKAY just no data and do not want to BIND
		521:  bytes_received:=0; //Connection has been refused by the remote host 
		523:  bytes_received:=0; //The host has not been found  
		524:  bytes_received:=0; //Host is unreachable  
		526:  bytes_received:=0; //The socket is not connected  
		527:  bytes_received:=0; //Shutdown has been called on the socket  
		529:  bytes_received:=0; //Socket has been gracefully closed. No more send/receives allowed	 
	END_CASE

	
	(*UDP: IPC returns -1 if no data available or error occured,841 returns -1 if error occured and 0 if no data available*)
	CASE bytes_received OF
	-2147483648..-1: ; (* No data available or error occured *)
	 0: IF NOT udp_mode OR pResult<>518 THEN (* TCP-Mode: socket wurde von remote geschlossen *)
			c_status := 253;
			c_ready := FALSE;
		END_IF;
	ELSE (* daten wurden empfangen *)
  		r_time := tx; (* Receive Timer ruecksetzen *)
		R_BUF.SIZE := INT_TO_UINT(r_offset) + DINT_TO_UINT(bytes_received); (* aktuelle buffersize eintragen *)
		IP_C.MAILBOX[1] := IP_C.MAILBOX[1] + 1; (* Receive Info *)
		IF IP_C.MAILBOX[1] = 0 THEN IP_C.MAILBOX[1] := 1; END_IF;

		(* ---------------------- Debug-Message ----------------------------*)
		(*IF _debug_enable THEN
			LOG_CL.NEW_MSG := 'IP_REC DATA: POS: ~1 : SIZE: ~2 TOTAL ~3 -IP_ID ~6';
			LOG_CL.PRINTF[1] := INT_TO_STRING(r_offset);
			LOG_CL.PRINTF[2] := INT_TO_STRING(r_count);
			LOG_CL.PRINTF[3] := UINT_TO_STRING(R_BUF.SIZE);
			LOG_CL.PRINTF[6] := INT_TO_STRING(debug_ID);
			LOG_MSG();
		END_IF;*)
		(* -----------------------------------------------------------------------------*)

	END_CASE
END_IF;

(* ---------------------------------------------- *)

IF S_BUF.SIZE > 0 THEN
	IF c_ready AND c_enable THEN
		IF NOT s_active AND IP_C.MAILBOX[2] = 0 THEN
			(* Gesamtanzahl an Bytes limitieren und uebergeben *)
			s_total := LIMIT(0,UINT_TO_INT(S_BUF.SIZE),r_max_size);
			s_cur_pos  := 0;
			s_cur_size := 0;
			s_start := TRUE; (* Daten kopieren und senden anstossen *)
			s_active := TRUE; (* Sende-Betrieb aktivieren *)
			(* ---------------------- Debug-Message ----------------------------*)
			(*IF _debug_enable THEN
				LOG_CL.NEW_MSG := 'IP_SEN INIT: TOTAL: ~1 -IP_ID ~6';
				LOG_CL.PRINTF[1] := INT_TO_STRING(S_TOTAL);
				LOG_CL.PRINTF[6] := INT_TO_STRING(debug_ID);
				LOG_MSG();
			END_IF;*)
			(* -----------------------------------------------------------------------------*)
		END_IF;

		IF s_done OR s_start THEN (* Daten senden aktiv *)

			s_start := FALSE;
			s_cur_pos := s_cur_pos + s_cur_size; (* neue Sende-Datenposition bestimmen *)
			IF s_total > s_cur_pos THEN (* weitere Daten zum senden vorhanden ? *)
				s_cur_size := s_total - s_cur_pos;
				s_cur_size := LIMIT(0, s_cur_size, s_max_size); (* Telegrammlänge begrenzen *)
				(* ---------------------- Debug-Message ----------------------------*)
				(*IF _debug_enable THEN
					LOG_CL.NEW_MSG := 'IP_SEN DATA: POS: ~1 : SIZE: ~2 TOTAL ~3 -IP_ID ~6';
					LOG_CL.PRINTF[1] := INT_TO_STRING(S_CUR_POS);
					LOG_CL.PRINTF[2] := INT_TO_STRING(S_CUR_SIZE);
					LOG_CL.PRINTF[3] := INT_TO_STRING(S_TOTAL);
					LOG_CL.PRINTF[6] := INT_TO_STRING(debug_ID);
					LOG_MSG();
				END_IF;*)
				(* -----------------------------------------------------------------------------*)
				s_time := tx; (* Send Timer ruecksetzen *)
				r_time := tx; (* Receive Timer ruecksetzen *)
				s_req := TRUE;

			ELSE
				(* keine weitere Sendedaten vorhanden -> Senden beenden *)
				s_req := FALSE;
				s_active := FALSE;
				S_BUF.SIZE := 0;
				(* ---------------------- Debug-Message ----------------------------*)
				(*IF _debug_enable THEN
					LOG_CL.NEW_MSG := 'IP_SEN FINISH -IP_ID ~6';
					LOG_CL.PRINTF[6] := INT_TO_STRING(debug_ID);
					LOG_MSG();
				END_IF;*)
				(* -----------------------------------------------------------------------------*)
			END_IF;
		END_IF;
	END_IF;
END_IF;

IF s_req THEN
	s_done := FALSE;
	IF udp_mode THEN
		bytes_sent := SysSockSendTo(socket, ADR(S_BUF.BUFFER[s_cur_pos]), s_cur_size, 0, ADR(sockaddr), SIZEOF(sockaddr), ADR(pResult));
	ELSE
		bytes_sent := SysSockSend(socket, ADR(S_BUF.BUFFER[s_cur_pos]), s_cur_size, 0, ADR(pResult));
	END_IF;

	CASE bytes_sent OF
	-2147483648..-1:	; (* ERROR: Noch nicht bereit um Daten aufzunehmen -> nächsten Zyklus wieder probieren *)
	 0: IF NOT udp_mode THEN (* TCP-Mode: socket wurde von remote geschlossen *)
			c_status := 253;
			c_ready := FALSE;
		END_IF;
	ELSE
		s_done := TRUE;
		s_cur_size := DINT_TO_INT(bytes_sent); (* Anzahl der wirklich versendeten Bytes übernehmen *)
		(* ---------------------- Debug-Message ----------------------------*)
		(*IF _debug_enable THEN
			LOG_CL.NEW_MSG := 'IP_SEN SEND_COUNT ~1 -IP_ID ~6';
			LOG_CL.PRINTF[1] := DINT_TO_STRING(s_cur_size);
			LOG_CL.PRINTF[6] := INT_TO_STRING(debug_ID);
			LOG_MSG();
		END_IF;*)
		(* -----------------------------------------------------------------------------*)
	END_CASE
END_IF;

(* ---------------------------------------------- *)

IF IP_C.R_OBSERVE = FALSE OR s_active THEN
    r_time := tx;
END_IF;

IF c_status = 0 AND tx - c_time > error_time AND c_enable AND NOT c_ready AND c_mode < 2 THEN (* Connect Timeout *)
	c_status := 255; (* Timeout-Fehler ausgeben *)
END_IF;
IF s_status = 0 AND tx - s_time > error_time AND s_active THEN (* Send Timeout *)
	s_status := 255; (* Timeout-Fehler ausgeben *)
END_IF;
IF r_status = 0 AND tx - r_time > error_time AND c_ready AND IP_C.R_OBSERVE THEN (* Receive Timeout *)
	r_status := 255; (* Timeout-Fehler ausgeben *)
END_IF;

IP_C.ERROR := DWORD_OF_BYTE(c_status,s_status,r_status,0);

(* ---------------------- Debug-Message ----------------------------*)
(*IF  _debug_enable THEN
	IF (IP_C.ERROR <> debug_lasterror) THEN
		LOG_CL.NEW_MSG := 'IP_ERROR ~1 -IP_ID ~6';
		LOG_CL.PRINTF[1] := DWORD_TO_STRING(IP_C.ERROR);
		LOG_CL.PRINTF[6] := INT_TO_STRING(debug_ID);
		LOG_MSG();

		debug_lasterror := IP_C.ERROR;
		debug_last_id := debug_ID;
	END_IF;
END_IF;*)
(* -----------------------------------------------------------------------------*)

(* revision history
ks	18. oct. 2008	rev 1.0
	original version
ks	05. jan. 2009	rev 1.1
	zusätzlichen Parameter "Port" hinzugefügt, und Code bei Verbindungsaufbau angepasst
ks	28. feb. 2009	rev 1.2
	connect code angepasst und verkürzung der zyklen bei Send
ks	20. oct. 2009	rev 1.3
	network_buffer basis 0
ks	06. dec. 2009	rev 1.4
	receive_count MAILBOX[1]
ks	10. nov. 2010	rev 1.5
	send_pause MAILBOX[2] and receive_pause MAILBOX[3] 
ks	07. feb. 2011	rev 1.6
	Fehlercode 253 bei Remote-Verbindungsabbruch
ks	30. may. 2011	rev 1.7
	Fehler bei Empfangsüberwachung
ks	26. july. 2011	rev 1.8
	Error-Reset, diverse optimierungen 
ks	26. feb. 2012	rev 1.9
	Code-Optimierung für höhere kompatibilität

*)

END_FUNCTION_BLOCK

// POUs/CONVERT/IP4_TO_STRING
FUNCTION IP4_TO_STRING : STRING(15)
VAR_INPUT
	IP4 : DWORD;
END_VAR
VAR
	tmp : STRING(3);
END_VAR

(*
version 1.1	10. mar. 2009
programmer 	kurt
tested by	hugo

IP4_TO_STRING erzeugt eine IP Adresse als String aus einem DWORD..

*)

(* mask bits AND INSERT AT given position *)
tmp := BYTE_TO_STRING(DWORD_TO_BYTE(IP4));
IP4_TO_STRING := CONCAT('...', tmp);
tmp := BYTE_TO_STRING(DWORD_TO_BYTE(SHR(IP4,8)));
IP4_TO_STRING := INSERT(IP4_TO_STRING, tmp, 2);
tmp := BYTE_TO_STRING(DWORD_TO_BYTE(SHR(IP4,16)));
IP4_TO_STRING := INSERT(IP4_TO_STRING, tmp, 1);
tmp := BYTE_TO_STRING(DWORD_TO_BYTE(SHR(IP4,24)));
IP4_TO_STRING := CONCAT(tmp, IP4_TO_STRING);



(* revision history
hm	22. apr 2008	rev 1.0
	original version

hm	10. mar. 2009	rev 1.1
	improved code
*)

END_FUNCTION

// POUs/NETWORK/LOG_MSG
FUNCTION_BLOCK LOG_MSG
(* VAR_EXTERNAL
	LOG_CL :	LOG_CONTROL;
END_VAR *)
VAR
	FB_PRINT_SF :PRINT_SF;
	idX : INT;
END_VAR

(*
version 1.0		01 mai 2010
programmer		ks
tested by		ks

LOG_MSG trägt Meldungen in den Loggingbuffer ein
*)

IF DWORD_TO_BYTE(SHL(LOG_CL.NEW_MSG_OPTION,16)) > LOG_CL.LEVEL THEN RETURN; END_IF; (* Logging freigegeben ?*)

FB_PRINT_SF(PRINTF_DATA := LOG_CL.PRINTF,STR := LOG_CL.NEW_MSG);

IF LOG_CL.RESET THEN (* Logeinträge löschen *)
	LOG_CL.RESET := FALSE;
	LOG_CL.RING_MODE := FALSE;
	LOG_CL.IDX := 0;
	LOG_CL.UPDATE_COUNT := LOG_CL.UPDATE_COUNT + UINT#1; (* UpdateCount erhöhen *)
END_IF;

IF LOG_CL.SIZE > 0 THEN (* size wert ist eingetragen *)
	IF LEN(LOG_CL.NEW_MSG) > 0 THEN (* Meldung in Puffer eintragen *)
		IF (LOG_CL.IDX >= LOG_CL.SIZE) THEN
			LOG_CL.RING_MODE := TRUE; (* bei Überlauf = Ringbuffermodus *)
			LOG_CL.IDX := 0; (* wieder auf arrayanfang positionieren *)
		END_IF;

		LOG_CL.UPDATE_COUNT := LOG_CL.UPDATE_COUNT + UINT#1; (* UpdateCount erhöhen *)
		LOG_CL.IDX := LOG_CL.IDX + INT#1; (* nächste freie Position *)
		idx := LOG_CL.IDX; (* lade aktuelle Log-Puffer Positition *)
		LOG_CL.MSG[idx] := LOG_CL.NEW_MSG; (* neuen Log-String in puffer ablegen  *)
		LOG_CL.MSG_OPTION[idx] := LOG_CL.NEW_MSG_OPTION; (* neue Log-String Option in puffer ablegen  *)
		LOG_CL.NEW_MSG := ''; (* letzten Log-String löschen *)
	END_IF;
END_IF;

END_FUNCTION_BLOCK

// POUs/NETWORK/PRINT_SF
FUNCTION_BLOCK PRINT_SF
VAR_IN_OUT
	PRINTF_DATA : PRINTF_DATA;
	STR : STRING(LOG_SIZE);
END_VAR
VAR
	pos : INT;
	c : INT;
	src : STRING(1) := '~';
	run : BOOL;
END_VAR

(*

version 1.0 		14. aug. 2009
programmer 	ks
tested by		ks

PRINTF erzeugt aus einem Parameterstring und den übergebenen Parameterdaten einen Text
*)

IF LEN(STR) > 0 THEN
	run := TRUE;

	WHILE (run) DO
		pos := FIND(STR,src);
		PRINTF_DATA[10] := '';

		IF pos = 0 THEN
			run:= FALSE;
		ELSE
			c := OSCAT_BASIC.CODE(STR:=STR,POS:=pos + 1);
			IF OSCAT_BASIC.ISC_NUM(INT_TO_BYTE(c)) THEN
				c := c - 48; (* notwendig weil innerhalb einer indexangabe nur eine var stehen darf *)
				PRINTF_DATA[10] := PRINTF_DATA[c]; (* Kommando 1-9 ergibt Parameterindex 1-9 *)
				(* Parameter gegen Text tauschen *)
			END_IF;
			IF LEN(PRINTF_DATA[10]) + LEN(STR) > LOG_SIZE THEN
				PRINTF_DATA[10] := '..';
			END_IF;
			(* pcworx: aus und eingangsstring muss verschieden sein *)
			PRINTF_DATA[11] := STR;
			STR := REPLACE(PRINTF_DATA[11],PRINTF_DATA[10],2,pos);
		END_IF;
	END_WHILE;
END_IF;

(* revision history

ks	14. aug. 2009	rev 1.0
	original version

*)

END_FUNCTION_BLOCK

// POUs/CONVERT/BASE64_DECODE_STR
FUNCTION_BLOCK BASE64_DECODE_STR
VAR_INPUT
	RUN : BOOL;
END_VAR
VAR_OUTPUT
	DONE : BOOL;
END_VAR
VAR_IN_OUT
	STR1 : STRING(192);
	STR2 : STRING(144);
END_VAR
VAR
	BASE64_DECODE_STREAM : BASE64_DECODE_STREAM;
	run_last : BOOL;
	buf1 : ARRAY [0..63] OF BYTE;
	buf2 : ARRAY [0..47] OF BYTE;
	mode : INT;
	size1 : INT;
	size2 : INT;
	end : INT;
	pos : INT;
END_VAR

(*
version 1.0	06. dec. 2009
programmer 	ks
tested by	ks

BASE64_DECODE_STR konvertiert einen BASE64 kodierten String in einen normalen String. 

*)

CASE mode OF
0:	IF RUN AND NOT run_last THEN
		DONE := FALSE;
		mode := 1;
		end := LEN(STR1);
		pos := 0;
		STR2 := '';
	END_IF;
1:
	size1 := MIN(48,end - pos);
	IF size1 > 0 THEN
		OSCAT_BASIC._STRING_TO_BUFFER(STR:=MID(STR1, size1, pos + 1), POS:=0, PT:=ADR(buf1), SIZE:=SIZEOF(buf1));
		BASE64_DECODE_STREAM(BUF1:=buf1 ,BUF2:=buf2 ,SIZE1:=size1 ,SIZE2=>size2);
		STR2 := CONCAT(STR2,OSCAT_BASIC.BUFFER_TO_STRING(PT:=ADR(buf2), SIZE:=SIZEOF(buf2), START:=0, STOP:=size2 - 1));
	ELSE
		mode := 0;
		DONE := TRUE;
	END_IF;
	pos := pos + size1;
END_CASE;

run_last := RUN;

(* revision history

ks	6. dec. 2009 rev 1.0
	original version

*)

END_FUNCTION_BLOCK

// POUs/CONVERT/BASE64_DECODE_STREAM
FUNCTION_BLOCK BASE64_DECODE_STREAM
VAR_IN_OUT
	BUF1 : ARRAY [0..63] OF BYTE;
	BUF2 : ARRAY [0..47] OF BYTE;
END_VAR
VAR_INPUT
	SIZE1 : INT;
END_VAR
VAR_OUTPUT
	SIZE2 : INT;
END_VAR
VAR_TEMP
	a: INT;
	b: WORD;
	o: INT;
	off: INT;
	i1: INT;
	i2: INT;
	c: INT;
END_VAR

(*
version 1.0	06. dec. 2009
programmer 	ks
tested by	ks

BASE64_DECODE_STREAM konvertiert einzelne Base64 kodierte Datenblöcke in normalen Datenblöcke. 

*)

IF SIZE1 <= 0 THEN SIZE2 := 0; RETURN; END_IF;
c := SIZE1 - 1;
i2 := 0;
a := 0;
b := 0;
FOR i1 := 0 TO c DO
	o := BUF1[i1];
	IF o = 61  (* = *) THEN	EXIT;
	ELSIF o > 96 (* a-z *) THEN off := 71;
	ELSIF o > 64 (* A-Z *) THEN off := 65;
	ELSIF o > 47 (* 0-9 *) THEN off := -4;
	ELSIF o = 43 (* + *) THEN off := -19;
	ELSIF o = 47 (* / *) THEN off := -16;
	END_IF;
	b := SHL(b,6) OR INT_TO_BYTE(o - off);
	a := a + 6;
	IF a >= 8 THEN
		a := a - 8;
		BUF2[i2] := WORD_TO_BYTE(SHR(b,a));
		i2 := i2 + 1;
		b := b AND NOT SHL(WORD#16#FFFF,a);
	END_IF;
END_FOR;
SIZE2 := i2;

(* revision history

ks	6. dec. 2009 rev 1.0
	original version

*)

END_FUNCTION_BLOCK

// POUs/CONVERT/BASE64_ENCODE_STR
FUNCTION_BLOCK BASE64_ENCODE_STR
VAR_INPUT
	RUN : BOOL;
END_VAR
VAR_OUTPUT
	DONE : BOOL;
END_VAR
VAR_IN_OUT
	STR1 : STRING(144);
	STR2 : STRING(192);
END_VAR
VAR
	BASE64_ENCODE_STREAM : BASE64_ENCODE_STREAM;
	run_last : BOOL;
	buf1 : ARRAY [0..47] OF BYTE;
	buf2 : ARRAY [0..63] OF BYTE;
	mode : INT;
	size1 : INT;
	size2 : INT;
	end : INT;
	pos : INT;
END_VAR

(*
version 1.0	06. dec. 2009
programmer 	ks
tested by	ks

BASE64_ENCODE_STR konvertiert einen normalen String in einen BASE64 kodierten String. 

*)

CASE mode OF
0:	IF RUN AND NOT run_last THEN
		DONE := FALSE;
		mode := 1;
		end := LEN(STR1);
		pos := 0;
		STR2 := '';
	END_IF;
1:
	size1 := MIN(48,end - pos);
	IF size1 > 0 THEN
		OSCAT_BASIC._STRING_TO_BUFFER(STR:=MID(STR1, size1, pos + 1), POS:=0, PT:=ADR(buf1), SIZE:=SIZEOF(buf1));
		BASE64_ENCODE_STREAM(BUF1:=buf1 ,BUF2:=buf2 ,SIZE1:=size1 ,SIZE2=>size2);
		STR2 := CONCAT(STR2,OSCAT_BASIC.BUFFER_TO_STRING(PT:=ADR(buf2), SIZE:=SIZEOF(buf2), START:=0, STOP:=size2 - 1));
	ELSE
		mode := 0;
		DONE := TRUE;
	END_IF;
	pos := pos + size1;
END_CASE;

run_last := RUN;

(* revision history

ks	6. dec. 2009 rev 1.0
	original version

*)

END_FUNCTION_BLOCK

// POUs/CONVERT/BASE64_ENCODE_STREAM
FUNCTION_BLOCK BASE64_ENCODE_STREAM
VAR_IN_OUT
	BUF1 : ARRAY [0..47] OF BYTE;
	BUF2 : ARRAY [0..63] OF BYTE;
END_VAR
VAR_INPUT
	SIZE1 : INT;
END_VAR
VAR_OUTPUT
	SIZE2 : INT;
END_VAR
VAR
	a: INT;
	b: WORD;
	i: INT;
	i2: INT;
	i3: INT;
	c: INT;
	BASE64: STRING(64) := 'ABCDEFGHIJKLMNOPQRSTUVWXYZabcdefghijklmnopqrstuvwxyz0123456789+/';
END_VAR

(*
version 1.0	06. dec. 2009
programmer 	ks
tested by	ks

BASE64_ENCODE_STREAM konvertiert Datenblöcke in Base64. 

*)

IF SIZE1 <= 0 THEN
	SIZE2 := 0;
	RETURN;
END_IF;
c := SIZE1 - 1;
i2 := 0;
a := 0;
b := 0;
FOR i := 0 TO c DO
	b := SHL(b,8) OR BUF1[i];
	a := a + 8;
	WHILE a >= 6 DO
		a := a - 6;
		buf2[i2] := OSCAT_BASIC.CODE(BASE64,WORD_TO_INT(SHR(b,a)) + 1);
		i2 := i2 + 1;
		b := b AND NOT SHL(WORD#16#FFFF,a);
	END_WHILE;
END_FOR;
IF a > 0 THEN
	buf2[i2] := OSCAT_BASIC.CODE(BASE64,WORD_TO_INT(SHL(b,6 - a)) + 1);
	i2 := i2 + 1;
	i3 := i2 + (NOT INT_TO_WORD(i2) AND 2#11);
	FOR i := i2 TO i3 DO
		buf2[i] := 61;
	END_FOR;
	SIZE2 := i3 + 1;
ELSE
	SIZE2 := i2;
END_IF;

(* revision history

ks	6. dec. 2009 rev 1.0
	original version

*)

END_FUNCTION_BLOCK

// POUs/FILE/CSV_PARSER_BUF
FUNCTION_BLOCK CSV_PARSER_BUF
VAR_INPUT
	SEP : BYTE;
END_VAR
VAR_IN_OUT
	RUN : BYTE;
	OFFSET : UDINT;
	VALUE : STRING(OSCAT_BASIC.STRING_LENGTH);
	PT : NETWORK_BUFFER;
END_VAR
VAR_OUTPUT
	RESULT : BYTE;
END_VAR
VAR
	step : INT;
	size : INT;
	c : BYTE;
	v_add : BYTE;
	i : INT;
	state : BYTE;
	eof : BOOL;
	pv : POINTER TO BYTE;
	pve : DWORD;
	watchdog : TON;
	x : BOOL;

	(*LOG_MSG : LOG_MSG;
	_debug_enable : BOOL := TRUE;
	step_last : INT;*)
END_VAR

(*
version 1.0		01. oct. 2010
programmer 		ks
tested by			ks

CSV_PARSER_BUF liefert die Elemente oder Zeilen einer Textdatei die in einem Bytearray abgelegt ist.

--------------------------------------

RUN Mode
00 = kein Befehl aktiv
01 = Element suchen

Result Codes
01 = Element gefunden
02 = Element und Zeilenende erkannt
05 = Befehl in Arbeit (Busy)
10 = nichts gefunden - Daten-Ende erreicht

State Codes
01 = Element gefunden
02 = Element und Zeilenende erkannt
05 = Befehl in Arbeit (Busy)
10 = nichts gefunden - Daten-Ende erreicht

*)

IF RUN > 0 THEN
	IF state = 0 THEN (* Auswertung neu beginnen *)

		pv := ADR(VALUE);
		pv^ := 0; (* VALUE = '' *)
		pve := pv + INT_TO_DWORD(OSCAT_BASIC.STRING_LENGTH);
		i := UDINT_TO_INT(OFFSET);
		size := UINT_TO_INT(PT.SIZE) - 1;
		RESULT := 0;
		state := 5; (* Befehl in Arbeit (Busy) *)
		step := 0; (* Auswertung neu beginnen *)

		(* ---------------- Debug-Message -----------------------*)
		(*IF _debug_enable THEN
			LOG_CL.NEW_MSG := 'CPF: Startindex: ~1';
			LOG_CL.PRINTF[1] := INT_TO_STRING(i);
			LOG_MSG();
		END_IF;*)
		(* -----------------------------------------------------------------*)

	END_IF;

	watchdog(IN:=FALSE,PT:=T#1ms); (* Timer neustarten *)
	watchdog.IN := TRUE;

	WHILE (state = 5) DO (* Schleife solange kein Ergebnis *)

		watchdog(); (* Timer aktualisieren *)

		IF watchdog.Q THEN (* watchdog ausgelöst *)
			state := 5;
			EXIT;
		ELSIF i > size THEN (* kein weiteres zeichen vorhanden *)
			state := 10; (* nichts gefunden - Daten-Ende erreicht *)
			EXIT;
		ELSE

			c := PT.BUFFER[i]; (* neues Zeichen aus Buffer lesen *)
			eof := i + 1 = PT.SIZE; (* End of File *)

			v_add := 0;

			IF c = SEP THEN (* Neues Element erkannt *)
				state := 1;
				x := TRUE;
			ELSIF c >= 32 THEN (* Element erkannt *)
				v_add := c; (* Zeichen ablegen *)
				IF eof THEN
					state := 2; (* Element und Zeilenende erkannt *)
				ELSE
					x := TRUE;
				END_IF;
			ELSE
				IF x THEN
					state := 2; (* Element und Zeilenende erkannt *)
					x := FALSE;
				END_IF;
			END_IF;

			IF v_add > 0  AND pv < pve THEN (* Zeichen zu Value-String hinzufügen *)
				pv^ := v_add; (* Zeichen eintragen *)
				pv := pv + 1;
				pv^ := 0; (* String-Terminierung eintragen *)
			END_IF;

			i := i + 1; (* Datenzeiger erhöhen *)

		END_IF;
	END_WHILE;

	CASE state OF
	01:	(* Element gefunden *)
		RESULT := 1; (* Element gefunden *)
		OFFSET := i; (* Offset uebernehmen *)
		RUN := 0;
		state := 0;
	02:	(* Element gefunden *)
		RESULT := 2; (* Element und Zeilenende erkannt *)
		OFFSET := i; (* Offset uebernehmen *)
		RUN := 0;
		state := 0;

	05:	RESULT := 5; (* in Arbeit *)

	10:	(* Indexüberschreitung - Bufferende *)
		RESULT := 10; (* nichts gefunden - Datenende erreicht *)
		OFFSET := i; (* Offset uebernehmen *)
		RUN := 0;
		state := 0;
	END_CASE;

	(* ---------------- Debug-Message -----------------------*)
	(*IF _debug_enable THEN
		LOG_CL.NEW_MSG := 'CPF: intern Result ~1 , state ~2, step ~3 , offset ~4, run ~5';
		LOG_CL.PRINTF[1] := BYTE_TO_STRING(RESULT);
		LOG_CL.PRINTF[2] := BYTE_TO_STRING(state);
		LOG_CL.PRINTF[3] := INT_TO_STRING(step);
		LOG_CL.PRINTF[4] := UDINT_TO_STRING(OFFSET);
		LOG_CL.PRINTF[5] := BYTE_TO_STRING(RUN);
		LOG_MSG();
	END_IF;*)
	(* -----------------------------------------------------------------*)

END_IF;

(* ---------------- Debug-Message -----------------------*)
(*IF _debug_enable THEN
	IF step_last <> step THEN
		LOG_CL.NEW_MSG := 'IPB: Step: ~1';
		LOG_CL.PRINTF[1]  := INT_TO_STRING(step);
		LOG_MSG();
	END_IF;
	step_last := step;
END_IF;*)
(* -----------------------------------------------------------------*)

(* revision history
ks	01. oct. 2010	rev 1.0
	original version
*)

END_FUNCTION_BLOCK

// POUs/DEMO/WORKING/INI_PARSER_BUF_DEMO
PROGRAM INI_PARSER_BUF_DEMO
VAR
	STATION_NAME : STRING;
	STATION_IP : STRING;
	SMTP_SERVER : STRING;
	SMTP_FROM :	STRING;

	IPB : INI_PARSER_BUF;
	FS : FILE_SERVER_V2;
	FSD : FILE_SERVER_DATA;
	PT : NETWORK_BUFFER;
	section : INT;
	key : STRING(OSCAT_BASIC.STRING_LENGTH);
	value : STRING(OSCAT_BASIC.STRING_LENGTH);
	str : STRING(OSCAT_BASIC.STRING_LENGTH);
	step : INT;
	result : BYTE;
	offset : UDINT;
	run : BYTE;
	done : BOOL;

	(*_debug_enable : BOOL := TRUE;
	LOG_MSG : LOG_MSG;*)
END_VAR

(* Demo-Programm: INI-Datei mittels Enumeration auswerten *)

(* ----- den nachfolgenden Textblock als datei "config.ini" auf der sps ablegen ---
# Demo - Initialisierungsdatei

[Station]
NAME=Test_Station_1
IP=192.168.178.1

[SMTP]
SERVER=test.server.de
FROM=test1@gmx.net
---------------------------------------------------------------------------------*)

CASE step OF

00:	IF NOT done THEN
	 	(* File_Daten einrichten  *)
		FSD.FILENAME := 'config.ini'; (* Dateiname *)
		FSD.MODE := 1; (* vorhandene Datei zum lesen öffnen *)
		FSD.OFFSET := 0; (* Start bei Dateianfang *)
		PT.SIZE := 65535; (* maximale länge einlesen *)
		step := 10;
	END_IF;

10:	IF FSD.MODE = 0 THEN (* Datei geöffnet ? *)
		OFFSET := 0; (* Start Offset vorgeben *)
		str := '';
		run := 3; (* key suchen *)
		step := 20;
	END_IF;

20:	IF run = 0 THEN
		(* ---------------------- Debug-Message ----------------------------*)
		(*IF _debug_enable THEN
			LOG_CL.NEW_MSG := 'IPBD: /key >~1< /value >~2< /offset ~3 /Run ~4 /Result ~5';
			LOG_CL.PRINTF[1] := key;
			LOG_CL.PRINTF[2] := value;
			LOG_CL.PRINTF[3] := UDINT_TO_STRING(OFFSET);
			LOG_CL.PRINTF[4] := BYTE_TO_STRING(run);
			LOG_CL.PRINTF[5] := BYTE_TO_STRING(result);
			LOG_MSG();
		END_IF;*)
		(* -----------------------------------------------------------------*)

		run := 3; (* vorbelegung -> naechsten key suchen *)

		IF result = 1 THEN (* neue Sektion gefunden *)
			IF key = 'Station' THEN
				section := 1;
			ELSIF key = 'SMTP' THEN
				section := 2;

			(* hier können weitere Section hinzugefügt werden *)

			ELSE
				section := 0; (* unbekannte sektion gefunden -> ignorieren *)
			END_IF;

		ELSIF result = 2 AND section > 0 THEN (* Key in einer bekannten sektion gefunden *)

			CASE section OF

			1:  (* Section: Station *)
				IF key = 'NAME' THEN
					STATION_NAME := value; (* Name *)
				ELSIF key = 'IP' THEN
					STATION_IP := value; (* IP-Adresse *)
				END_IF;

				(* hier können weitere Schlüsselsauswertungen hinzugefügt werden *)

			2:  (* Section: SMTP *)
				IF key = 'SERVER' THEN
					SMTP_SERVER := value; (* SMTP Server *)
				ELSIF key = 'FROM' THEN
					SMTP_FROM := value; (* SMTP Absender *)
				END_IF;

				(* hier können weitere Schlüsselsauswertungen hinzugefügt werden *)

			END_CASE;

		ELSIF result = 10 THEN (* nichts mehr gefunden *)
			run := 0; (* keine weitere INI Auswertung erwünscht *)
			FSD.MODE := 5; (* Datei schliessen *)
			step := 30;
		END_IF;
	END_IF;

30:	IF FSD.MODE = 0 THEN (* Datei geschlossen ? *)
		step := 0;
		done := TRUE;
	END_IF;

END_CASE;

IPB(STR:=str,RUN:=run,OFFSET:=OFFSET,KEY:=key,VALUE:=value,PT:=PT); (* INI PARAMETER BUF *)
result:=IPB.RESULT;

FS(FSD:=FSD,PT:=PT); (* FILE_SERVER *)

END_PROGRAM

// POUs/_HARDWARE/FILE_SERVER
FUNCTION_BLOCK FILE_SERVER
VAR_IN_OUT
	FSD : FILE_SERVER_DATA;
	PT : NETWORK_BUFFER;
END_VAR
VAR
	buf_size : UDINT;
	handle : DWORD;
	read_max_length : UDINT;
	file_position : UDINT;
	used_filename : STRING;
	close_time : TIME;
	length_read : UDINT;
	write_length : UDINT;
	length_written : UDINT;
	open_handle : DWORD;
	seek_position : UDINT;
	tell_position : UDINT;
	file_size : UDINT;
	open_mode : STRING(2);
	open_AccessMode :  UDINT;
	last_mode: BYTE;
	command : BYTE;
	error_code : BYTE;
	error : BOOL;
	file_change : BOOL;
	step : INT;
	t_diff : TIME;
	tx : TIME;
	tx_last : TIME;

	(*step_last : INT;
	FB_LOG_MESSAGE : LOG_MSG;
	_debug_enable : BOOL := TRUE;*)
	COMMAND_DELAY_TON: TON;
	pResult : UDINT;
END_VAR
(*
version 1.0	20. apr. 2010
programmer 	ks
tested by		ks

FILE_SERVER ermöglicht den Zugriff auf Dateien mittels Plattform-Neutraler Schnittstelle
*)

(*
1 = File_Open_Exist + File_Read
2 = File_Open_Exist + File_Write
3 = File_Open_New   + File_Write
4 = File_Remove
5 = File_Close

- Action -
1 = file_open   (open)
2 = file_close  (close)
3 = file_read   (read)
4 = file_write  (write)
5 = file_seek   (setpos)
6 = file_tell   (getpos)
7 = file_remove (delete)

---- fehlermeldungen----

0						Kein Fehler
1	SysFileOpen		Fehler
2	SysFileClose		Fehler
3	SysFileRead		Fehler
4	SysFileWrite		Fehler
5	SysFileSetPos	Fehler
6	SysFileGetPos	Fehler
7	SysFileDelete		Fehler
8	SysFileGetSize	Fehler
255	Applikation	Position liegt hinter dem Dateiende

*)

CASE step OF
0:
	IF FSD.MODE = LIMIT(1,FSD.MODE,5) THEN

		(* ---------------------- Debug-Message ----------------------------*)
		(*IF _debug_enable THEN
			LOG_CL.NEW_MSG := 'File_Start Mode=~1';
			LOG_CL.PRINTF[1] := BYTE_TO_STRING(FSD.MODE);
			FB_LOG_MESSAGE();
		END_IF;*)
		(* -----------------------------------------------------------------*)

		buf_size := SIZEOF(PT.BUFFER);

		IF FSD.MODE = 4 THEN (* File_Remove *)
			IF handle > 0 THEN
				File_change := TRUE;
				step := 32000; (* File_Close ausführen *)
			ELSE
				step := 90; (* File_Remove ausführen *)
			END_IF;

		ELSIF FSD.MODE = 5 THEN (* File_Close *)
			step := 32000; (* File_Close ausführen *)

		ELSIF handle = 0 THEN (* MODE 1,2,3 *)
			step := 100; (* File muss erst geöffnet werden *)

		ELSE (* File ist geöffnset *)
			IF used_filename = FSD.FILENAME AND FSD.MODE = last_mode THEN (* kein Moduswechsel ? *)
				step := 200; (* ohne open prozedure weitermachen *)
			ELSE
				step := 32000;
				File_change := TRUE;
			END_IF;
		END_IF;
	END_IF;

(* ----------------------------------- *)
090: (* File_Remove *)
	command := 7; (* File Remove *)
	step := 95;

095: (* File_Remove beendet *)
	IF command = 0 THEN
		step := 30000; (* Beenden *)
	END_IF;
(* ----------------------------------- *)

100: (* File Size - Dateigroesse bestimmen *)
	command := 8; (* File Size *)
	step := 110;

110: (* File Size beendet *)
	IF command = 0 THEN
		IF FSD.MODE = 1 THEN (* open + read *)
			open_mode := 'r';
			open_AccessMode:=AM_READ_PLUS;
			FSD.FILE_SIZE := file_size; (* aktuelle Dateigroesse *)
		ELSIF FSD.MODE = 2 THEN (* open + write *)
			open_mode := 'a';
			open_AccessMode:=AM_APPEND_PLUS;
			FSD.FILE_SIZE := file_size; (* aktuelle Dateigroesse *)
		ELSE (* open new + write *)
			open_mode := 'w';
			open_AccessMode:=AM_WRITE_PLUS;
			FSD.FILE_SIZE := 0; (* aktuelle Dateigroesse *)
		END_IF;
		command := 1; (* File Open *)
		last_mode := FSD.MODE;
		step := 150; (* File_Open ausführen *)
	END_IF;

150: (* File Open *)
	IF command = BYTE#0 THEN
		IF error THEN
			step := 30000; (* Beenden *)
		ELSE
			(* Filedaten eintragen *)
			handle := open_handle;
			used_filename := FSD.FILENAME;
			file_position := UDINT#4294967295; (* maximal = unbekannt *)
			FSD.FILE_OPEN := TRUE;
			step := 200;
		END_IF;
	END_IF;

200: (* File Seek *)
	IF FSD.OFFSET = UDINT#4294967294 THEN (* 16#FFFF_FFFE -> Zeiger auf Dateiende stellen *)
		command := 5; (* File-Seek *)
		seek_position := FSD.FILE_SIZE;
		step := 210;
	ELSIF FSD.OFFSET > FSD.FILE_SIZE THEN (* prüfe auf gültige offset-vorgabe *)
		error_code := 255;
		step := 30000; (* Beenden *)
	ELSIF FSD.OFFSET <> file_position THEN
		command := 5; (* File-Seek *)
		seek_position := FSD.OFFSET;
		step := 210;
	ELSE
		step := 300;
	END_IF;

210: (* File Seek *)
	IF command = 0 THEN
		file_position := seek_position;
		IF error THEN
			step := 30000; (* Beenden *)
		ELSE
			step := 300;
		END_IF;
	END_IF;

300: (* Read or Write ? *)
	IF FSD.MODE = 1 THEN
		step := 400; (* Read *)
	ELSE
		step := 500; (* Write *)
	END_IF;

400: (* File Read *)
	IF UINT_TO_UDINT(PT.SIZE) > buf_size THEN (* Leselänge auf Buffergroesse begrenzen *)
		read_max_length := buf_size;
	ELSE
		read_max_length := UINT_TO_UDINT(PT.SIZE);
	END_IF;

	(* Leselänge an Dateilänge anpassen *)
	IF file_position + read_max_length > FSD.FILE_SIZE THEN
		read_max_length := FSD.FILE_SIZE - file_position;
	END_IF;

	IF read_max_length > 0 THEN
		command := 3; (* File_Read *)
		step := 410;
	ELSE
		PT.SIZE := UINT#0;
		step := 30000; (* Beenden *)
	END_IF;

410: (* File Read *)
	IF command = 0 THEN
		PT.SIZE := UDINT_TO_UINT(length_read);
		IF NOT Error THEN
			file_position := file_position + length_read; (* aktueller File_Position korrigieren *)
			FSD.OFFSET := file_position;
		END_IF;
		step := 30000; (* Beenden *)
	END_IF;

500: (* File Write *)
	IF UINT_TO_UDINT(PT.SIZE) > buf_size THEN (* Schreiblänge auf Buffergroesse begrenzen *)
		write_length := buf_size;
	ELSE
		write_length := UINT_TO_UDINT(PT.SIZE);
	END_IF;

	IF write_length > 0 THEN
		command := 4; (* File_Write *)
		step := 510;
	ELSE
		step := 30000; (* Beenden *)
	END_IF;

510:
	IF command = 0 THEN
		IF NOT Error THEN
			file_position := file_position + length_written; (* aktueller File_Position korrigieren *)
			FSD.OFFSET := file_position;
			IF file_position > FSD.FILE_SIZE THEN (* Datei ist groesser geworden *)
				FSD.FILE_SIZE := file_position;
			END_IF;
		END_IF;
		step := 30000; (* Beenden *)
	END_IF;

 (* --------------------------------------------- *)

30000: (* Befehl fertig *)
	FSD.MODE := 0;
	FSD.ERROR := error_code;
	step := 0;

	(* ---------------- Debug-Message -----------------------*)
	(*IF _debug_enable THEN
		LOG_CL.NEW_MSG := 'File_Stop: File ~1, error ~7, code ~8';
		LOG_CL.PRINTF[1]  := used_filename;
		LOG_CL.PRINTF[7]  := INT_TO_STRING(BOOL_TO_INT(error));
		LOG_CL.PRINTF[8]  := BYTE_TO_STRING(error_code);
		FB_LOG_MESSAGE();
	END_IF;*)
	(* --------------------------------------------- *)

32000:
	IF handle > 0 THEN
		command := 2; (* File_Close ausführen *)
	END_IF;
	step := 32100;

32100:
	IF command = 0 THEN (* File Close beendet *)
		(* Filedaten ablöschen *)
		FSD.FILE_OPEN := FALSE;
		file_position := 0;
		FSD.FILE_SIZE := 0;
		FSD.OFFSET := 0;
		used_filename := '';
		handle := 0;

		(* File_Name wurde fliegend geändert ? *)
		IF File_change THEN
			File_change := FALSE;
			step := 0;
		ELSE
			step := 30000;
		END_IF;
	END_IF;

END_CASE;

(* 1 = file_open
   2 = file_close
   3 = file_read
   4 = file_write
   5 = file_seek
   6 = file_tell
   7 = file_remove
*) 

(* ------------ File Open ------------- *)
IF command = 1 THEN
	open_handle := SysFileOpen(FSD.FILENAME,open_AccessMode, ADR(pResult) );
	error := open_handle = 0 OR open_handle = 16#FFFFFFFF;
	error_code := SEL(error,0,command);
	command := 0;

	(* ---------------- Debug-Message -----------------------*)
	(*IF _debug_enable THEN
		LOG_CL.NEW_MSG := 'Open: File ~1, handle ~2 , mode ~3 , error ~7, code ~8';
		LOG_CL.PRINTF[1] := FSD.FILENAME;
		LOG_CL.PRINTF[2] := DWORD_TO_STRING(open_handle);
		LOG_CL.PRINTF[3] := open_mode;
		LOG_CL.PRINTF[7] := INT_TO_STRING(BOOL_TO_INT(error));
		LOG_CL.PRINTF[8] := BYTE_TO_STRING(error_code);
		FB_LOG_MESSAGE();
	END_IF;*)
	(* -----------------------------------------------------------------*)
END_IF;

(* ----------- File Close ------------- *)
IF command = 2 THEN
	error := NOT SysFileClose(handle)=0;
	error_code := SEL(error,0,command);
	command := 0;

	(* ---------------- Debug-Message -----------------------*)
	(*IF _debug_enable THEN
		LOG_CL.NEW_MSG := 'Close: File ~1, error ~7, code ~8';
		LOG_CL.PRINTF[1] := used_filename;
		LOG_CL.PRINTF[7] := INT_TO_STRING(BOOL_TO_INT(error));
		LOG_CL.PRINTF[8] := BYTE_TO_STRING(error_code);
		FB_LOG_MESSAGE();
	END_IF;*)
	(* -----------------------------------------------------------------*)
END_IF;

(* ------------ File Read ------------- *)
IF command = 3 THEN
	length_read := SysFileRead(handle, ADR(PT.BUFFER), read_max_length, ADR(pResult) );
	error := length_read = 0;
	error_code := SEL(error,0,command);
	command := 0;

	(* ---------------- Debug-Message -----------------------*)
	(*IF _debug_enable THEN
		LOG_CL.NEW_MSG := 'Read: File ~1, soll ~2,ist ~3 ,error ~7, code ~8';
		LOG_CL.PRINTF[1] := used_filename;
		LOG_CL.PRINTF[2] := UDINT_TO_STRING(read_max_length);
		LOG_CL.PRINTF[3] := UDINT_TO_STRING(length_read);
		LOG_CL.PRINTF[7] := INT_TO_STRING(BOOL_TO_INT(error));
		LOG_CL.PRINTF[8] := BYTE_TO_STRING(error_code);
		FB_LOG_MESSAGE();
	END_IF;*)
	(* -----------------------------------------------------------------*)
END_IF;

(* ------------ File Write ------------- *)
IF command = 4 THEN
	length_written := SysFileWrite(handle, ADR(PT.BUFFER), write_length, ADR(pResult) );
	error := length_written = 0;
	error_code := SEL(error,0,command);
	command := 0;

	(* ---------------- Debug-Message -----------------------*)
	(*IF _debug_enable THEN
		LOG_CL.NEW_MSG := 'Write: File ~1, soll ~2,ist ~3 ,error ~7, code ~8';
		LOG_CL.PRINTF[1] := used_filename;
		LOG_CL.PRINTF[2] := UDINT_TO_STRING(write_length);
		LOG_CL.PRINTF[3] := UDINT_TO_STRING(length_written);
		LOG_CL.PRINTF[7] := INT_TO_STRING(BOOL_TO_INT(error));
		LOG_CL.PRINTF[8] := BYTE_TO_STRING(error_code);
		FB_LOG_MESSAGE();
	END_IF;*)
	(* -----------------------------------------------------------------*)
END_IF;

(* ------------ File Seek ------------- *)
IF command = 5 THEN
	error := NOT SysFileSetPos(handle, seek_position)=0;
	error_code := SEL(error,0,command);
	command := 0;

	(* ---------------- Debug-Message -----------------------*)
	(*IF _debug_enable THEN
		LOG_CL.NEW_MSG := 'Seek: File ~1,pos ~3 ,error ~7, code ~8';
		LOG_CL.PRINTF[1] := used_filename;
		LOG_CL.PRINTF[3] := UDINT_TO_STRING(seek_position);
		LOG_CL.PRINTF[7] := INT_TO_STRING(BOOL_TO_INT(error));
		LOG_CL.PRINTF[8] := BYTE_TO_STRING(error_code);
		FB_LOG_MESSAGE();
	END_IF;*)
	(* -----------------------------------------------------------------*)
END_IF;

(* ------------ File Tell ------------- *)
IF command = 6 THEN
	tell_position := SysFileGetPos(handle, ADR(pResult) );
	error := tell_position < 0;
	error_code := SEL(error,0,command);
	command := 0;

	(* ---------------- Debug-Message -----------------------*)
	(*IF _debug_enable THEN
		LOG_CL.NEW_MSG := 'Tell: File ~1, pos ~3 ,error ~7, code ~8';
		LOG_CL.PRINTF[1] := used_filename;
		LOG_CL.PRINTF[3] := UDINT_TO_STRING(tell_position);
		LOG_CL.PRINTF[7] := INT_TO_STRING(BOOL_TO_INT(error));
		LOG_CL.PRINTF[8] := BYTE_TO_STRING(error_code);
		FB_LOG_MESSAGE();
	END_IF;*)
	(* -----------------------------------------------------------------*)
END_IF;

(* ------------ File Remove ------------- *)
IF command = 7 THEN
	error := NOT SysFileDelete(FSD.FILENAME)=0;
	error_code := SEL(error,0,command);
	command := 0;

	(* ---------------- Debug-Message -----------------------*)
	(*IF _debug_enable THEN
		LOG_CL.NEW_MSG := 'Remove: File ~1, error ~7, code ~8';
		LOG_CL.PRINTF[1] := FSD.FILENAME;
		LOG_CL.PRINTF[7] := INT_TO_STRING(BOOL_TO_INT(error));
		LOG_CL.PRINTF[8] := BYTE_TO_STRING(error_code);
		FB_LOG_MESSAGE();
	END_IF;*)
	(* -----------------------------------------------------------------*)
END_IF;

(* ------------ File Size ------------- *)
IF command = 8 THEN
	file_size := SysFileGetSize(FSD.FILENAME, ADR(pResult) );
	error_code := 0; (* kein Errorcode vorhanden *)
	command := 0;

	(* ---------------- Debug-Message -----------------------*)
	(*IF _debug_enable THEN
		LOG_CL.NEW_MSG := 'Size: File ~1, size ~3, error ~7, code ~8';
		LOG_CL.PRINTF[1] := FSD.FILENAME;
		LOG_CL.PRINTF[3] := DINT_TO_STRING(file_size);
		LOG_CL.PRINTF[7] := INT_TO_STRING(BOOL_TO_INT(error));
		LOG_CL.PRINTF[8] := BYTE_TO_STRING(error_code);
		FB_LOG_MESSAGE();
	END_IF;*)
	(* -----------------------------------------------------------------*)
END_IF;

(* ---------------- Debug-Message -----------------------*)
(*IF _debug_enable THEN
	IF step_last <> step THEN
		LOG_CL.NEW_MSG := 'Step: ~1';
		LOG_CL.PRINTF[1] := INT_TO_STRING(step);
		FB_LOG_MESSAGE();
	END_IF;
	step_last := step;
END_IF;*)
(* -----------------------------------------------------------------*)

(* revision history
ks	05. mai. 2012	rev 1.1
	auto_close funktion entfernt

ks	23. sep. 2010	rev 1.0
	original version
*)

END_FUNCTION_BLOCK

// POUs/FILE/INI_PARSER_BUF
FUNCTION_BLOCK INI_PARSER_BUF
VAR_IN_OUT
	STR : STRING(OSCAT_BASIC.STRING_LENGTH);
	RUN : BYTE;
	OFFSET : UDINT;
	KEY : STRING(OSCAT_BASIC.STRING_LENGTH);
	VALUE : STRING(OSCAT_BASIC.STRING_LENGTH);
	PT : NETWORK_BUFFER;
END_VAR
VAR_OUTPUT
	RESULT : BYTE;
END_VAR
VAR
	step : INT;
	size : INT;
	c : BYTE;
	k_add : BYTE;
	v_add : BYTE;
	i : INT;
	state : BYTE;
	eof : BOOL;
	pv : POINTER TO BYTE;
	pk : POINTER TO BYTE;
	pve : DWORD;
	pke : DWORD;
	watchdog : TON;

	(*LOG_MSG : LOG_MSG;
	_debug_enable : BOOL := TRUE;
	step_last : INT;*)
END_VAR

(*
version 1.0		23. sep. 2010
programmer 		ks
tested by			ks

INI_PARSER_BUF liefert die Elemente einer Initialisierungsdatei die in einem Bytearray abgelegt ist.

--------------------------------------

RUN Mode
00 = kein Befehl aktiv
01 = Section melden
02 = Key melden
03 = Section oder Key melden

Result Codes
01 = Section gefunden
02 = Key gefunden
05 = Befehl in Arbeit (Busy)
10 = nichts gefunden - Daten-Ende erreicht
11 = keinen Key gefunden - Section-Ende erreicht

State Codes
00 = Indexüberschreitung - Bufferende
01 = Section gefunden
02 = Key gefunden
03 = Kommentar gefunden
05 = Befehl in Arbeit (Busy)
10 = nichts gefunden - Daten-Ende erreicht

*)

IF RUN > 0 THEN
	IF state = 0 THEN (* Auswertung neu beginnen *)

		pv := ADR(VALUE);
		pv^ := 0; (* VALUE = '' *)
		pve := pv + INT_TO_DWORD(OSCAT_BASIC.STRING_LENGTH);
		pk := ADR(KEY);
		pk^ := 0; (* KEY = '' *)
		pke := pk + INT_TO_DWORD(OSCAT_BASIC.STRING_LENGTH);

		i := UDINT_TO_INT(OFFSET);
		size := UINT_TO_INT(PT.SIZE) - 1;
		RESULT := 0;
		state := 5; (* Befehl in Arbeit (Busy) *)
		step := 0; (* Auswertung neu beginnen *)

		(*####################  DEBUG-MESSAGE  ###################################*)
		(*IF _debug_enable THEN
			LOG_CL.NEW_MSG := 'IPB: Startindex: ~1';
			LOG_CL.PRINTF[1]  := INT_TO_STRING(i);
			LOG_MSG();
		END_IF;*)
		(*########################################################################*)
	END_IF;

	watchdog(IN:=FALSE,PT:=T#1ms); (* Timer neustarten *)
	watchdog.IN := TRUE;

	WHILE (state = 5) DO (* Schleife solange kein Ergebnis *)

		watchdog(); (* Timer aktualisieren *)

		IF watchdog.Q THEN (* watchdog ausgelöst *)
			state := 5;
			EXIT;
		ELSIF i > size THEN (* kein weiteres zeichen vorhanden *)
			state := 10; (* nichts gefunden - Daten-Ende erreicht *)
			EXIT;
		ELSE

			c := PT.BUFFER[i]; (* neues Zeichen aus Buffer lesen *)
			eof := i + 1 = PT.SIZE; (* End of File *)

			k_add := 0;
			v_add := 0;

			CASE step OF

			0: (* noch kein Modus erkannt *)
				IF c = 91 THEN (* mit "[" vergleichen *)
					step := 200; (* Modus für Section aktivieren *)
				ELSIF c = 59 OR c = 35 THEN (* mit ";" und '#' vergleichen *)
					step := 100; (* Modus für Kommentar aktivieren *)
				ELSIF c > 32 THEN (* Key erkannt *)
					k_add := c; (* Zeichen ablegen *)
					step := 300; (* Key auswertung starten *)
				END_IF;
			100: (* Kommentar erkannt -> Zeilenende suchen *)
				IF c < 32 THEN (* prüfe auf Steuerzeichen *)
					state  := 3; (* Beenden -> Kommentar wurde gefunden *)
				END_IF;
			200: (* Sections-start erkannt -> Sectionsende suchen *)
				IF c = 93 THEN (* mit "]" vergleichen *)
					IF pk > ADR(KEY) > 0 THEN (* innerhalb von [] muss sich mindestens ein Zeichen befinden *)
						state  := 1; (* Beenden -> Section wurde gefunden *)
					ELSE
						pk := ADR(KEY);
						pk^ := 0; (* KEY = '' *)
						step := 0; (* fehlerhafte Section-Zeile vorhanden -> weitersuchen *)
					END_IF;
				ELSIF c < 32 OR eof THEN (* Steuerzeichen - fehlerhafte Section-Zeile -> weitersuchen *)
					pk := ADR(KEY);
					pk^ := 0; (* KEY = '' *)
					step := 0;
				ELSE
					k_add := c; (* Zeichen ablegen *)
				END_IF;
			300: (* Beginn: Key erkannt -> Name auswerten *)
				IF c < 32 THEN (* Steuerzeichen - fehlerhafte Key-Zeile -> weitersuchen *)
					pk := ADR(KEY);
					pk^ := 0; (* KEY = '' *)
					step := 0;
				ELSIF c = 61 THEN (* prüfe auf '=' *)
					step := 330;
				ELSE
					k_add := c; (* Zeichen ablegen *)
				END_IF;
			330: (* KeyValue beginn suchen *)
				IF c < 32 THEN (* Steuerzeichen  *)
					state := 2; (* Key ohne Value gefunden *)
				ELSIF eof THEN
					state := 2; (* Key ohne Value gefunden *)
					v_add := c; (* Zeichen ablegen *)
				ELSE
					v_add := c; (* Zeichen ablegen *)
					step := 350;
				END_IF;
			350: (* KeyValue Ende suchen *)
				IF c < 32 THEN (* Steuerzeichen *)
					state := 2; (* Key gefunden *)
				ELSIF eof THEN
					v_add := c; (* Zeichen ablegen *)
					state := 2; (* Key gefunden *)
				ELSE
					v_add := c; (* Zeichen ablegen *)
				END_IF;
			END_CASE;

			IF v_add > 0  AND pv < pve THEN (* Zeichen zu Value-String hinzufügen *)
				pv^ := v_add; (* Zeichen eintragen *)
				pv := pv + 1;
				pv^ := 0; (* String-Terminierung eintragen *)
			END_IF;

			IF k_add > 0 AND pk < pke THEN (* Zeichen zu Key-String hinzufügen *)
				pk^ := k_add; (* Zeichen eintragen *)
				pk := pk + 1;
				pk^ := 0; (* String-Terminierung eintragen *)
			END_IF;

			i := i + 1; (* Datenzeiger erhöhen *)

		END_IF;
	END_WHILE;

	CASE state OF
	01:	(* Section gefunden *)
		IF RUN = 1 OR RUN = 3 THEN (* Section vorgewählt oder alles rückmelden *)
			IF KEY = STR OR LEN(STR) = 0 THEN (* mit gesuchter Section vergleichen oder keine Section vorgegeben *)
				RESULT := 1; (* Section gefunden *)
				OFFSET := i; (* Offset uebernehmen *)
				RUN := 0;
				state := 0;
			END_IF;
		ELSE
			pk := ADR(KEY);
			pk^ := 0; (* KEY = '' *)
			RESULT := 11; (* Key nicht gefunden , Section-Ende - Offset nicht verändern *)
			RUN := 0;
			state := 0;
		END_IF;
	02:	(* Key gefunden *)
		IF RUN = 2 OR RUN = 3 THEN (* Key vorgewählt oder alles rückmelden *)
			IF KEY = STR OR LEN(STR) = 0 THEN (* mit gesuchten Key vergleichen *)
				RESULT := 2; (* Key gefunden *)
				OFFSET := i; (* Offset uebernehmen *)
				RUN := 0;
				state := 0;
			END_IF;
		END_IF;
	03:	(* Kommenar gefunden *)
		OFFSET := i; (* Offset uebernehmen *)
		state := 0;

	05:	RESULT := 5; (* in Arbeit *)

	10:	(* Indexüberschreitung - Bufferende *)
		RESULT := 10; (* nichts gefunden - Datenende erreicht *)
		OFFSET := i; (* Offset uebernehmen *)
		RUN := 0;
		state := 0;
	END_CASE;

	(*####################  DEBUG-MESSAGE  ###################################*)
	(*IF _debug_enable THEN
		LOG_CL.NEW_MSG := 'IPF: intern Result ~1 , state ~2, step ~3 , offset ~4, run ~5';
		LOG_CL.PRINTF[1] := BYTE_TO_STRING(RESULT);
		LOG_CL.PRINTF[2] := BYTE_TO_STRING(state);
		LOG_CL.PRINTF[3] := INT_TO_STRING(step);
		LOG_CL.PRINTF[4] := UDINT_TO_STRING(OFFSET);
		LOG_CL.PRINTF[5] := BYTE_TO_STRING(RUN);
		LOG_MSG();
	END_IF;*)
	(*########################################################################*)

END_IF;

(*####################  DEBUG-MESSAGE  ###################################*)
(*IF _debug_enable THEN
	IF step_last <> step THEN
		LOG_CL.NEW_MSG := 'IPB: Step: ~1';
		LOG_CL.PRINTF[1]  := INT_TO_STRING(step);
		LOG_MSG();
	END_IF;
	step_last := step;
END_IF;*)
(*########################################################################*)

(* revision history
ks	23. sep. 2010	rev 1.0
	original version
*)

END_FUNCTION_BLOCK

// POUs/HARDWARE/FILE_SERVER_V2
FUNCTION_BLOCK FILE_SERVER_V2
VAR_IN_OUT
	FSD : FILE_SERVER_DATA;
	PT : NETWORK_BUFFER;
END_VAR
VAR
	buf_size : UDINT;
	handle : DWORD;
	read_max_length : UDINT;
	file_position : UDINT;
	used_filename : STRING;
	length_read : UDINT;
	write_length : UDINT;
	length_written : UDINT;
	open_handle : DWORD;
	seek_position : UDINT;
	tell_position : UDINT;
	file_size : DINT;
	open_mode : STRING(2);
	last_mode: BYTE;
	command : BYTE;
	error_code : BYTE;
	error : BOOL;
	file_change : BOOL;
	step : INT;

	(*step_last : INT;
	FB_LOG_MESSAGE : LOG_MSG;
	_debug_enable : BOOL := TRUE;*)
END_VAR
(*
version 1.1	05. mai. 2012
programmer 	ks
tested by		ks

FILE_SERVER ermöglicht den Zugriff auf Dateien mittels Plattform-Neutraler Schnittstelle
*)

(*
1 = File_Open_Exist + File_Read
2 = File_Open_Exist + File_Write
3 = File_Open_New   + File_Write
4 = File_Remove
5 = File_Close

- Action -
1 = file_open   (open)
2 = file_close  (close)
3 = file_read   (read)
4 = file_write  (write)
5 = file_seek   (setpos)
6 = file_tell   (getpos)
7 = file_remove (delete)

---- fehlermeldungen----

0						Kein Fehler
1	SysFileOpen		Fehler
2	SysFileClose		Fehler
3	SysFileRead		Fehler
4	SysFileWrite		Fehler
5	SysFileSetPos	Fehler
6	SysFileGetPos	Fehler
7	SysFileDelete		Fehler
8	SysFileGetSize	Fehler
255	Applikation	Position liegt hinter dem Dateiende

*)

CASE step OF
0:
	IF FSD.MODE = LIMIT(1,FSD.MODE,5) THEN

		(* ---------------------- Debug-Message ----------------------------*)
		(*IF _debug_enable THEN
			LOG_CL.NEW_MSG := 'File_Start Mode=~1';
			LOG_CL.PRINTF[1] := BYTE_TO_STRING(FSD.MODE);
			FB_LOG_MESSAGE();
		END_IF;*)
		(* -----------------------------------------------------------------*)

		buf_size := SIZEOF(PT.BUFFER);

		IF FSD.MODE = 4 THEN (* File_Remove *)
			IF handle > 0 THEN
				File_change := TRUE;
				step := 32000; (* File_Close ausführen *)
			ELSE
				step := 90; (* File_Remove ausführen *)
			END_IF;

		ELSIF FSD.MODE = 5 THEN (* File_Close *)
			step := 32000; (* File_Close ausführen *)

		ELSIF handle = 0 THEN (* MODE 1,2,3 *)
			step := 100; (* File muss erst geöffnet werden *)

		ELSE (* File ist geöffnset *)
			IF used_filename = FSD.FILENAME AND FSD.MODE = last_mode THEN (* kein Moduswechsel ? *)
				step := 200; (* ohne open prozedure weitermachen *)
			ELSE
				step := 32000;
				File_change := TRUE;
			END_IF;
		END_IF;
	END_IF;

(* ----------------------------------- *)
090: (* File_Remove *)
	command := 7; (* File Remove *)
	step := 95;

095: (* File_Remove beendet *)
	IF command = 0 THEN
		step := 30000; (* Beenden *)
	END_IF;
(* ----------------------------------- *)

100: (* File Size - Dateigroesse bestimmen *)
	command := 8; (* File Size *)
	step := 110;

110: (* File Size beendet *)
	IF command = 0 THEN
		IF FSD.MODE = 1 THEN (* open + read *)
			open_mode := 'r';
			FSD.FILE_SIZE := file_size; (* aktuelle Dateigroesse *)
		ELSIF FSD.MODE = 2 THEN (* open + write *)
			open_mode := 'a';
			FSD.FILE_SIZE := file_size; (* aktuelle Dateigroesse *)
		ELSE (* open new + write *)
			open_mode := 'w';
			FSD.FILE_SIZE := 0; (* aktuelle Dateigroesse *)
		END_IF;
		command := 1; (* File Open *)
		last_mode := FSD.MODE;
		step := 150; (* File_Open ausführen *)
	END_IF;

150: (* File Open *)
	IF command = BYTE#0 THEN
		IF error THEN
			step := 30000; (* Beenden *)
		ELSE
			(* Filedaten eintragen *)
			handle := open_handle;
			used_filename := FSD.FILENAME;
			file_position := UDINT#4294967295; (* maximal = unbekannt *)
			FSD.FILE_OPEN := TRUE;
			step := 200;
		END_IF;
	END_IF;

200: (* File Seek *)
	IF FSD.OFFSET = UDINT#4294967294 THEN (* 16#FFFF_FFFE -> Zeiger auf Dateiende stellen *)
		command := 5; (* File-Seek *)
		seek_position := FSD.FILE_SIZE;
		step := 210;
	ELSIF FSD.OFFSET > FSD.FILE_SIZE THEN (* prüfe auf gültige offset-vorgabe *)
		error_code := 255;
		step := 30000; (* Beenden *)
	ELSIF FSD.OFFSET <> file_position THEN
		command := 5; (* File-Seek *)
		seek_position := FSD.OFFSET;
		step := 210;
	ELSE
		step := 300;
	END_IF;

210: (* File Seek *)
	IF command = 0 THEN
		file_position := seek_position;
		IF error THEN
			step := 30000; (* Beenden *)
		ELSE
			step := 300;
		END_IF;
	END_IF;

300: (* Read or Write ? *)
	IF FSD.MODE = 1 THEN
		step := 400; (* Read *)
	ELSE
		step := 500; (* Write *)
	END_IF;

400: (* File Read *)
	IF UINT_TO_UDINT(PT.SIZE) > buf_size THEN (* Leselänge auf Buffergroesse begrenzen *)
		read_max_length := buf_size;
	ELSE
		read_max_length := UINT_TO_UDINT(PT.SIZE);
	END_IF;

	(* Leselänge an Dateilänge anpassen *)
	IF file_position + read_max_length > FSD.FILE_SIZE THEN
		read_max_length := FSD.FILE_SIZE - file_position;
	END_IF;

	IF read_max_length > 0 THEN
		command := 3; (* File_Read *)
		step := 410;
	ELSE
		PT.SIZE := UINT#0;
		step := 30000; (* Beenden *)
	END_IF;

410: (* File Read *)
	IF command = 0 THEN
		PT.SIZE := UDINT_TO_UINT(length_read);
		IF NOT Error THEN
			file_position := file_position + length_read; (* aktueller File_Position korrigieren *)
			FSD.OFFSET := file_position;
		END_IF;
		step := 30000; (* Beenden *)
	END_IF;

500: (* File Write *)
	IF UINT_TO_UDINT(PT.SIZE) > buf_size THEN (* Schreiblänge auf Buffergroesse begrenzen *)
		write_length := buf_size;
	ELSE
		write_length := UINT_TO_UDINT(PT.SIZE);
	END_IF;

	IF write_length > 0 THEN
		command := 4; (* File_Write *)
		step := 510;
	ELSE
		step := 30000; (* Beenden *)
	END_IF;

510:
	IF command = 0 THEN
		IF NOT Error THEN
			file_position := file_position + length_written; (* aktueller File_Position korrigieren *)
			FSD.OFFSET := file_position;
			IF file_position > FSD.FILE_SIZE THEN (* Datei ist groesser geworden *)
				FSD.FILE_SIZE := file_position;
			END_IF;
		END_IF;
		step := 30000; (* Beenden *)
	END_IF;

 (* --------------------------------------------- *)

30000: (* Befehl fertig *)
	FSD.MODE := 0;
	FSD.ERROR := error_code;
	step := 0;

	(* ---------------- Debug-Message -----------------------*)
	(*IF _debug_enable THEN
		LOG_CL.NEW_MSG := 'File_Stop: File ~1, error ~7, code ~8';
		LOG_CL.PRINTF[1]  := used_filename;
		LOG_CL.PRINTF[7]  := INT_TO_STRING(BOOL_TO_INT(error));
		LOG_CL.PRINTF[8]  := BYTE_TO_STRING(error_code);
		FB_LOG_MESSAGE();
	END_IF;*)
	(* --------------------------------------------- *)

32000:
	IF handle > 0 THEN
		command := 2; (* File_Close ausführen *)
	END_IF;
	step := 32100;

32100:
	IF command = 0 THEN (* File Close beendet *)
		(* Filedaten ablöschen *)
		FSD.FILE_OPEN := FALSE;
		file_position := 0;
		FSD.FILE_SIZE := 0;
		FSD.OFFSET := 0;
		used_filename := '';
		handle := 0;

		(* File_Name wurde fliegend geändert ? *)
		IF File_change THEN
			File_change := FALSE;
			step := 0;
		ELSE
			step := 30000;
		END_IF;
	END_IF;

END_CASE;

(* 1 = file_open
   2 = file_close
   3 = file_read
   4 = file_write
   5 = file_seek
   6 = file_tell
   7 = file_remove
*) 

(* ------------ File Open ------------- *)
IF command = 1 THEN
	open_handle := SysFileOpen(FSD.FILENAME,open_mode);
	error := open_handle = 0;
	error_code := SEL(error,0,command);
	command := 0;

	(* ---------------- Debug-Message -----------------------*)
	(*IF _debug_enable THEN
		LOG_CL.NEW_MSG := 'Open: File ~1, handle ~2 , mode ~3 , error ~7, code ~8';
		LOG_CL.PRINTF[1] := FSD.FILENAME;
		LOG_CL.PRINTF[2] := DWORD_TO_STRING(open_handle);
		LOG_CL.PRINTF[3] := open_mode;
		LOG_CL.PRINTF[7] := INT_TO_STRING(BOOL_TO_INT(error));
		LOG_CL.PRINTF[8] := BYTE_TO_STRING(error_code);
		FB_LOG_MESSAGE();
	END_IF;*)
	(* -----------------------------------------------------------------*)
END_IF;

(* ----------- File Close ------------- *)
IF command = 2 THEN
	error := NOT SysFileClose(handle);
	error_code := SEL(error,0,command);
	command := 0;

	(* ---------------- Debug-Message -----------------------*)
	(*IF _debug_enable THEN
		LOG_CL.NEW_MSG := 'Close: File ~1, error ~7, code ~8';
		LOG_CL.PRINTF[1] := used_filename;
		LOG_CL.PRINTF[7] := INT_TO_STRING(BOOL_TO_INT(error));
		LOG_CL.PRINTF[8] := BYTE_TO_STRING(error_code);
		FB_LOG_MESSAGE();
	END_IF;*)
	(* -----------------------------------------------------------------*)
END_IF;

(* ------------ File Read ------------- *)
IF command = 3 THEN
	length_read := SysFileRead(handle, ADR(PT.BUFFER), read_max_length);
	error := length_read = 0;
	error_code := SEL(error,0,command);
	command := 0;

	(* ---------------- Debug-Message -----------------------*)
	(*IF _debug_enable THEN
		LOG_CL.NEW_MSG := 'Read: File ~1, soll ~2,ist ~3 ,error ~7, code ~8';
		LOG_CL.PRINTF[1] := used_filename;
		LOG_CL.PRINTF[2] := UDINT_TO_STRING(read_max_length);
		LOG_CL.PRINTF[3] := UDINT_TO_STRING(length_read);
		LOG_CL.PRINTF[7] := INT_TO_STRING(BOOL_TO_INT(error));
		LOG_CL.PRINTF[8] := BYTE_TO_STRING(error_code);
		FB_LOG_MESSAGE();
	END_IF;*)
	(* -----------------------------------------------------------------*)
END_IF;

(* ------------ File Write ------------- *)
IF command = 4 THEN
	length_written := SysFileWrite(handle, ADR(PT.BUFFER), write_length);
	error := length_written = 0;
	error_code := SEL(error,0,command);
	command := 0;

	(* ---------------- Debug-Message -----------------------*)
	(*IF _debug_enable THEN
		LOG_CL.NEW_MSG := 'Write: File ~1, soll ~2,ist ~3 ,error ~7, code ~8';
		LOG_CL.PRINTF[1] := used_filename;
		LOG_CL.PRINTF[2] := UDINT_TO_STRING(write_length);
		LOG_CL.PRINTF[3] := UDINT_TO_STRING(length_written);
		LOG_CL.PRINTF[7] := INT_TO_STRING(BOOL_TO_INT(error));
		LOG_CL.PRINTF[8] := BYTE_TO_STRING(error_code);
		FB_LOG_MESSAGE();
	END_IF;*)
	(* -----------------------------------------------------------------*)
END_IF;

(* ------------ File Seek ------------- *)
IF command = 5 THEN
	error := NOT SysFileSetPos(handle, seek_position);
	error_code := SEL(error,0,command);
	command := 0;

	(* ---------------- Debug-Message -----------------------*)
	(*IF _debug_enable THEN
		LOG_CL.NEW_MSG := 'Seek: File ~1,pos ~3 ,error ~7, code ~8';
		LOG_CL.PRINTF[1] := used_filename;
		LOG_CL.PRINTF[3] := UDINT_TO_STRING(seek_position);
		LOG_CL.PRINTF[7] := INT_TO_STRING(BOOL_TO_INT(error));
		LOG_CL.PRINTF[8] := BYTE_TO_STRING(error_code);
		FB_LOG_MESSAGE();
	END_IF;*)
	(* -----------------------------------------------------------------*)
END_IF;

(* ------------ File Tell ------------- *)
IF command = 6 THEN
	tell_position := SysFileGetPos(handle);
	error := tell_position < 0;
	error_code := SEL(error,0,command);
	command := 0;

	(* ---------------- Debug-Message -----------------------*)
	(*IF _debug_enable THEN
		LOG_CL.NEW_MSG := 'Tell: File ~1, pos ~3 ,error ~7, code ~8';
		LOG_CL.PRINTF[1] := used_filename;
		LOG_CL.PRINTF[3] := UDINT_TO_STRING(tell_position);
		LOG_CL.PRINTF[7] := INT_TO_STRING(BOOL_TO_INT(error));
		LOG_CL.PRINTF[8] := BYTE_TO_STRING(error_code);
		FB_LOG_MESSAGE();
	END_IF;*)
	(* -----------------------------------------------------------------*)
END_IF;

(* ------------ File Remove ------------- *)
IF command = 7 THEN
	error := NOT SysFileDelete(FSD.FILENAME);
	error_code := SEL(error,0,command);
	command := 0;

	(* ---------------- Debug-Message -----------------------*)
	(*IF _debug_enable THEN
		LOG_CL.NEW_MSG := 'Remove: File ~1, error ~7, code ~8';
		LOG_CL.PRINTF[1] := FSD.FILENAME;
		LOG_CL.PRINTF[7] := INT_TO_STRING(BOOL_TO_INT(error));
		LOG_CL.PRINTF[8] := BYTE_TO_STRING(error_code);
		FB_LOG_MESSAGE();
	END_IF;*)
	(* -----------------------------------------------------------------*)
END_IF;

(* ------------ File Size ------------- *)
IF command = 8 THEN
	file_size := SysFileGetSize(FSD.FILENAME);
	error_code := 0; (* kein Errorcode vorhanden *)
	command := 0;

	(* ---------------- Debug-Message -----------------------*)
	(*IF _debug_enable THEN
		LOG_CL.NEW_MSG := 'Size: File ~1, size ~3, error ~7, code ~8';
		LOG_CL.PRINTF[1] := FSD.FILENAME;
		LOG_CL.PRINTF[3] := DINT_TO_STRING(file_size);
		LOG_CL.PRINTF[7] := INT_TO_STRING(BOOL_TO_INT(error));
		LOG_CL.PRINTF[8] := BYTE_TO_STRING(error_code);
		FB_LOG_MESSAGE();
	END_IF;*)
	(* -----------------------------------------------------------------*)
END_IF;

(* ---------------- Debug-Message -----------------------*)
(*IF _debug_enable THEN
	IF step_last <> step THEN
		LOG_CL.NEW_MSG := 'Step: ~1';
		LOG_CL.PRINTF[1] := INT_TO_STRING(step);
		FB_LOG_MESSAGE();
	END_IF;
	step_last := step;
END_IF;*)
(* -----------------------------------------------------------------*)

(* revision history
ks	05. mai. 2012	rev 1.1
	auto_close funktion entfernt

ks	23. sep. 2010	rev 1.0
	original version
*)

END_FUNCTION_BLOCK

